LIN {X 0,Y 523.533,Z 695.705,A -85,B 0,C 180,E1 -4777.714,E2 -4777.714} C_VEL
LIN {X 0,Y 523.698,Z 688.725,A -85,B 0,C 180,E1 -4779.266,E2 -4779.266} C_VEL
LIN {X 0,Y 523.966,Z 679.973,A -85,B 0,C 180,E1 -4780.822,E2 -4780.822} C_VEL
LIN {X 0,Y 524.199,Z 670.632,A -85,B 0,C 180,E1 -4782.193,E2 -4782.193} C_VEL
LIN {X 0,Y 524.547,Z 661.185,A -85,B 0,C 180,E1 -4783.362,E2 -4783.362} C_VEL
LIN {X 0,Y 524.925,Z 649.916,A -85,B 0,C 180,E1 -4784.537,E2 -4784.537} C_VEL
LIN {X 0,Y 525.405,Z 637.565,A -85,B 0,C 180,E1 -4785.614,E2 -4785.614} C_VEL
LIN {X 0,Y 525.852,Z 623.929,A -85,B 0,C 180,E1 -4786.598,E2 -4786.598} C_VEL
LIN {X 0,Y 526.332,Z 610.529,A -85,B 0,C 180,E1 -4787.382,E2 -4787.382} C_VEL
LIN {X 0,Y 526.758,Z 595.819,A -85,B 0,C 180,E1 -4788.07,E2 -4788.07} C_VEL
LIN {X 0,Y 527.136,Z 580.489,A -85,B 0,C 180,E1 -4788.61,E2 -4788.61} C_VEL
LIN {X 0,Y 527.421,Z 564.422,A -85,B 0,C 180,E1 -4788.998,E2 -4788.998} C_VEL
LIN {X 0,Y 528.018,Z 482.561,A -85,B 0,C 180,E1 -4790.169,E2 -4790.169} C_VEL
LIN {X 0,Y 528.423,Z 411.771,A -85,B 0,C 180,E1 -4791.166,E2 -4791.166} C_VEL
LIN {X 0,Y 525.812,Z 398.27,A -85,B 0,C 180,E1 -4791.495,E2 -4791.495} C_VEL
LIN {X 0,Y 526.43,Z 378.923,A -85,B 0,C 180,E1 -4794.026,E2 -4794.026} C_VEL
LIN {X 0,Y 526.914,Z 363.166,A -85,B 0,C 180,E1 -4796.112,E2 -4796.112} C_VEL
LIN {X 0,Y 523.93,Z 349.852,A -85,B 0,C 180,E1 -4798.108,E2 -4798.108} C_VEL
LIN {X 0,Y 523.931,Z 349.846,A -85,B 0,C 180,E1 -4800.852,E2 -4800.852} C_VEL
LIN {X 0,Y 523.922,Z 349.847,A -85,B 0,C 180,E1 -4803.728,E2 -4803.728} C_VEL
LIN {X 0,Y 523.878,Z 349.856,A -85,B 0,C 180,E1 -4806.398,E2 -4806.398} C_VEL
LIN {X 0,Y 523.901,Z 349.847,A -85,B 0,C 180,E1 -4809.084,E2 -4809.084} C_VEL
LIN {X 0,Y 523.899,Z 349.854,A -85,B 0,C 180,E1 -4812.122,E2 -4812.122} C_VEL
LIN {X 0,Y 523.922,Z 349.843,A -85,B 0,C 180,E1 -4815.31,E2 -4815.31} C_VEL
LIN {X 0,Y 523.907,Z 349.847,A -85,B 0,C 180,E1 -4818.693,E2 -4818.693} C_VEL
LIN {X 0,Y 523.889,Z 349.852,A -85,B 0,C 180,E1 -4821.896,E2 -4821.896} C_VEL
LIN {X 0,Y 523.902,Z 349.845,A -85,B 0,C 180,E1 -4824.912,E2 -4824.912} C_VEL
LIN {X 0,Y 523.921,Z 349.846,A -85,B 0,C 180,E1 -4827.679,E2 -4827.679} C_VEL
LIN {X 0,Y 523.92,Z 349.845,A -85,B 0,C 180,E1 -4830.68,E2 -4830.68} C_VEL
LIN {X 0,Y 523.883,Z 349.851,A -85,B 0,C 180,E1 -4833.724,E2 -4833.724} C_VEL
LIN {X 0,Y 523.892,Z 349.853,A -85,B 0,C 180,E1 -4836.269,E2 -4836.269} C_VEL
LIN {X 0,Y 523.924,Z 349.843,A -85,B 0,C 180,E1 -4838.766,E2 -4838.766} C_VEL
LIN {X 0,Y 523.918,Z 349.843,A -85,B 0,C 180,E1 -4841.22,E2 -4841.22} C_VEL
LIN {X 0,Y 523.897,Z 349.85,A -85,B 0,C 180,E1 -4844.437,E2 -4844.437} C_VEL
LIN {X 0,Y 523.937,Z 349.844,A -85,B 0,C 180,E1 -4847.607,E2 -4847.607} C_VEL
LIN {X 0,Y 523.914,Z 349.852,A -85,B 0,C 180,E1 -4849.957,E2 -4849.957} C_VEL
LIN {X 0,Y 523.975,Z 349.836,A -85,B 0,C 180,E1 -4853.067,E2 -4853.067} C_VEL
LIN {X 0,Y 523.934,Z 349.842,A -85,B 0,C 180,E1 -4855.384,E2 -4855.384} C_VEL
LIN {X 0,Y 524.089,Z 349.826,A -85,B 0,C 180,E1 -4857.695,E2 -4857.695} C_VEL
LIN {X 0,Y 524.081,Z 349.832,A -85,B 0,C 180,E1 -4860,E2 -4860} C_VEL
LIN {X 0,Y 524.088,Z 349.826,A -85,B 0,C 180,E1 -4862.306,E2 -4862.306} C_VEL
LIN {X 0,Y 523.991,Z 349.841,A -85,B 0,C 180,E1 -4866.16,E2 -4866.16} C_VEL
LIN {X 0,Y 523.96,Z 349.839,A -85,B 0,C 180,E1 -4869.263,E2 -4869.263} C_VEL
LIN {X 0,Y 523.931,Z 349.844,A -85,B 0,C 180,E1 -4872.394,E2 -4872.394} C_VEL
LIN {X 0,Y 523.898,Z 349.849,A -85,B 0,C 180,E1 -4875.563,E2 -4875.563} C_VEL
LIN {X 0,Y 523.914,Z 349.844,A -85,B 0,C 180,E1 -4878.781,E2 -4878.781} C_VEL
LIN {X 0,Y 523.925,Z 349.843,A -85,B 0,C 180,E1 -4881.234,E2 -4881.234} C_VEL
LIN {X 0,Y 523.918,Z 349.848,A -85,B 0,C 180,E1 -4884.197,E2 -4884.197} C_VEL
LIN {X 0,Y 523.879,Z 349.848,A -85,B 0,C 180,E1 -4887.137,E2 -4887.137} C_VEL
LIN {X 0,Y 523.882,Z 349.855,A -85,B 0,C 180,E1 -4889.76,E2 -4889.76} C_VEL
LIN {X 0,Y 523.921,Z 349.844,A -85,B 0,C 180,E1 -4892.451,E2 -4892.451} C_VEL
LIN {X 0,Y 523.897,Z 349.847,A -85,B 0,C 180,E1 -4895.229,E2 -4895.229} C_VEL
LIN {X 0,Y 523.891,Z 349.852,A -85,B 0,C 180,E1 -4898.104,E2 -4898.104} C_VEL
LIN {X 0,Y 523.907,Z 349.846,A -85,B 0,C 180,E1 -4901.307,E2 -4901.307} C_VEL
LIN {X 0,Y 523.925,Z 349.842,A -85,B 0,C 180,E1 -4904.69,E2 -4904.69} C_VEL
LIN {X 0,Y 523.878,Z 349.848,A -85,B 0,C 180,E1 -4906.88,E2 -4906.88} C_VEL
LIN {X 0,Y 523.194,Z 349.94,A -85,B 0,C 180,E1 -4907.521,E2 -4907.521} C_VEL
LIN {X 0,Y 520.328,Z 350.292,A -85,B 0,C 180,E1 -4908.563,E2 -4908.563} C_VEL
LIN {X 0,Y 517.929,Z 350.592,A -85,B 0,C 180,E1 -4909.401,E2 -4909.401} C_VEL
LIN {X 0,Y 516.921,Z 350.72,A -85,B 0,C 180,E1 -4910.049,E2 -4910.049} C_VEL
LIN {X 0,Y 516.85,Z 350.726,A -85,B 0,C 180,E1 -4910.269,E2 -4910.269} C_VEL
LIN {X 0,Y 516.839,Z 350.728,A -85,B 0,C 180,E1 -4913.349,E2 -4913.349} C_VEL
LIN {X 0,Y 516.878,Z 350.724,A -85,B 0,C 180,E1 -4916.12,E2 -4916.12} C_VEL
LIN {X 0,Y 516.884,Z 350.719,A -85,B 0,C 180,E1 -4918.938,E2 -4918.938} C_VEL
LIN {X 0,Y 516.837,Z 350.732,A -85,B 0,C 180,E1 -4921.582,E2 -4921.582} C_VEL
LIN {X 0,Y 516.866,Z 350.724,A -85,B 0,C 180,E1 -4924.209,E2 -4924.209} C_VEL
LIN {X 0,Y 516.855,Z 350.723,A -85,B 0,C 180,E1 -4926.777,E2 -4926.777} C_VEL
LIN {X 0,Y 516.938,Z 350.722,A -85,B 0,C 180,E1 -4929.733,E2 -4929.733} C_VEL
LIN {X 0,Y 516.883,Z 350.719,A -85,B 0,C 180,E1 -4932.596,E2 -4932.596} C_VEL
LIN {X 0,Y 516.936,Z 350.714,A -85,B 0,C 180,E1 -4935.031,E2 -4935.031} C_VEL
LIN {X 0,Y 516.968,Z 350.711,A -85,B 0,C 180,E1 -4938.235,E2 -4938.235} C_VEL
LIN {X 0,Y 516.932,Z 350.718,A -85,B 0,C 180,E1 -4941.4,E2 -4941.4} C_VEL
LIN {X 0,Y 516.987,Z 350.707,A -85,B 0,C 180,E1 -4944.541,E2 -4944.541} C_VEL
LIN {X 0,Y 517.077,Z 350.705,A -85,B 0,C 180,E1 -4947.664,E2 -4947.664} C_VEL
LIN {X 0,Y 517.069,Z 350.7,A -85,B 0,C 180,E1 -4950.001,E2 -4950.001} C_VEL
LIN {X 0,Y 517.077,Z 350.696,A -85,B 0,C 180,E1 -4952.338,E2 -4952.338} C_VEL
LIN {X 0,Y 516.979,Z 350.709,A -85,B 0,C 180,E1 -4956.245,E2 -4956.245} C_VEL
LIN {X 0,Y 516.94,Z 350.718,A -85,B 0,C 180,E1 -4959.391,E2 -4959.391} C_VEL
LIN {X 0,Y 516.958,Z 350.716,A -85,B 0,C 180,E1 -4961.808,E2 -4961.808} C_VEL
LIN {X 0,Y 516.949,Z 350.714,A -85,B 0,C 180,E1 -4965.146,E2 -4965.146} C_VEL
LIN {X 0,Y 516.882,Z 350.721,A -85,B 0,C 180,E1 -4968.225,E2 -4968.225} C_VEL
LIN {X 0,Y 516.911,Z 350.716,A -85,B 0,C 180,E1 -4970.703,E2 -4970.703} C_VEL
LIN {X 0,Y 516.89,Z 350.721,A -85,B 0,C 180,E1 -4974.074,E2 -4974.074} C_VEL
LIN {X 0,Y 516.849,Z 350.724,A -85,B 0,C 180,E1 -4976.663,E2 -4976.663} C_VEL
LIN {X 0,Y 516.892,Z 350.727,A -85,B 0,C 180,E1 -4979.519,E2 -4979.519} C_VEL
LIN {X 0,Y 516.902,Z 350.717,A -85,B 0,C 180,E1 -4982.544,E2 -4982.544} C_VEL
LIN {X 0,Y 516.867,Z 350.728,A -85,B 0,C 180,E1 -4985.329,E2 -4985.329} C_VEL
LIN {X 0,Y 516.884,Z 350.724,A -85,B 0,C 180,E1 -4987.943,E2 -4987.943} C_VEL
LIN {X 0,Y 516.878,Z 350.723,A -85,B 0,C 180,E1 -4990.743,E2 -4990.743} C_VEL
LIN {X 0,Y 516.887,Z 350.727,A -85,B 0,C 180,E1 -4993.893,E2 -4993.893} C_VEL
LIN {X 0,Y 516.924,Z 350.853,A -85,B 0,C 180,E1 -4996.033,E2 -4996.033} C_VEL
LIN {X 0,Y 518.959,Z 360.312,A -85,B 0,C 180,E1 -4997.639,E2 -4997.639} C_VEL
LIN {X 0,Y 518.787,Z 370.855,A -85,B 0,C 180,E1 -4999.267,E2 -4999.267} C_VEL
LIN {X 0,Y 521.906,Z 385.017,A -85,B 0,C 180,E1 -4999.622,E2 -4999.622} C_VEL
LIN {X 0,Y 520.71,Z 536.608,A -85,B 0,C 180,E1 -5001.836,E2 -5001.836} C_VEL
LIN {X 0,Y 520.403,Z 552.083,A -85,B 0,C 180,E1 -5002.224,E2 -5002.224} C_VEL
LIN {X 0,Y 519.996,Z 566.356,A -85,B 0,C 180,E1 -5002.733,E2 -5002.733} C_VEL
LIN {X 0,Y 519.561,Z 580.137,A -85,B 0,C 180,E1 -5003.38,E2 -5003.38} C_VEL
LIN {X 0,Y 519.167,Z 592.322,A -85,B 0,C 180,E1 -5004.09,E2 -5004.09} C_VEL
LIN {X 0,Y 518.645,Z 604.733,A -85,B 0,C 180,E1 -5004.955,E2 -5004.955} C_VEL
LIN {X 0,Y 518.169,Z 617.851,A -85,B 0,C 180,E1 -5006.069,E2 -5006.069} C_VEL
LIN {X 0,Y 517.742,Z 628.127,A -85,B 0,C 180,E1 -5007.113,E2 -5007.113} C_VEL
LIN {X 0,Y 517.366,Z 637.65,A -85,B 0,C 180,E1 -5008.238,E2 -5008.238} C_VEL
LIN {X 0,Y 517.032,Z 647.144,A -85,B 0,C 180,E1 -5009.579,E2 -5009.579} C_VEL
LIN {X 0,Y 516.749,Z 655.098,A -85,B 0,C 180,E1 -5010.908,E2 -5010.908} C_VEL
LIN {X 0,Y 516.536,Z 662.608,A -85,B 0,C 180,E1 -5012.444,E2 -5012.444} C_VEL
LIN {X 0,Y 516.42,Z 668.488,A -85,B 0,C 180,E1 -5013.923,E2 -5013.923} C_VEL
LIN {X 0,Y 516.306,Z 673.209,A -85,B 0,C 180,E1 -5015.455,E2 -5015.455} C_VEL
LIN {X 0,Y 516.214,Z 676.291,A -85,B 0,C 180,E1 -5016.745,E2 -5016.745} C_VEL
LIN {X 0,Y 516.181,Z 678.984,A -85,B 0,C 180,E1 -5018.431,E2 -5018.431} C_VEL
LIN {X 0,Y 516.199,Z 680.402,A -85,B 0,C 180,E1 -5020.1,E2 -5020.1} C_VEL
LIN {X 0,Y 516.165,Z 680.465,A -85,B 0,C 180,E1 -5021.75,E2 -5021.75} C_VEL
LIN {X 0,Y 516.169,Z 679.334,A -85,B 0,C 180,E1 -5023.385,E2 -5023.385} C_VEL
LIN {X 0,Y 516.212,Z 676.933,A -85,B 0,C 180,E1 -5025.008,E2 -5025.008} C_VEL
LIN {X 0,Y 516.279,Z 673.27,A -85,B 0,C 180,E1 -5026.619,E2 -5026.619} C_VEL
LIN {X 0,Y 516.387,Z 668.327,A -85,B 0,C 180,E1 -5028.22,E2 -5028.22} C_VEL
LIN {X 0,Y 516.557,Z 661.89,A -85,B 0,C 180,E1 -5029.812,E2 -5029.812} C_VEL
LIN {X 0,Y 516.8,Z 653.92,A -85,B 0,C 180,E1 -5031.397,E2 -5031.397} C_VEL
LIN {X 0,Y 517.106,Z 645.168,A -85,B 0,C 180,E1 -5032.817,E2 -5032.817} C_VEL
LIN {X 0,Y 517.457,Z 635.233,A -85,B 0,C 180,E1 -5034.153,E2 -5034.153} C_VEL
LIN {X 0,Y 517.851,Z 624.884,A -85,B 0,C 180,E1 -5035.329,E2 -5035.329} C_VEL
LIN {X 0,Y 518.291,Z 613.595,A -85,B 0,C 180,E1 -5036.404,E2 -5036.404} C_VEL
LIN {X 0,Y 518.823,Z 601.429,A -85,B 0,C 180,E1 -5037.379,E2 -5037.379} C_VEL
LIN {X 0,Y 519.301,Z 588.182,A -85,B 0,C 180,E1 -5038.255,E2 -5038.255} C_VEL
LIN {X 0,Y 519.79,Z 573.497,A -85,B 0,C 180,E1 -5039.031,E2 -5039.031} C_VEL
LIN {X 0,Y 520.184,Z 558.316,A -85,B 0,C 180,E1 -5039.648,E2 -5039.648} C_VEL
LIN {X 0,Y 520.543,Z 542.685,A -85,B 0,C 180,E1 -5040.103,E2 -5040.103} C_VEL
LIN {X 0,Y 520.711,Z 526.129,A -85,B 0,C 180,E1 -5040.409,E2 -5040.409} C_VEL
LIN {X 0,Y 521.891,Z 388.15,A -85,B 0,C 180,E1 -5042.421,E2 -5042.421} C_VEL
LIN {X 0,Y 521.675,Z 383.753,A -85,B 0,C 180,E1 -5042.499,E2 -5042.499} C_VEL
LIN {X 0,Y 518.92,Z 371.346,A -85,B 0,C 180,E1 -5042.821,E2 -5042.821} C_VEL
LIN {X 0,Y 519.16,Z 360.873,A -85,B 0,C 180,E1 -5044.464,E2 -5044.464} C_VEL
LIN {X 0,Y 517.011,Z 350.712,A -85,B 0,C 180,E1 -5046.243,E2 -5046.243} C_VEL
LIN {X 0,Y 516.942,Z 350.718,A -85,B 0,C 180,E1 -5049.389,E2 -5049.389} C_VEL
LIN {X 0,Y 516.957,Z 350.713,A -85,B 0,C 180,E1 -5051.807,E2 -5051.807} C_VEL
LIN {X 0,Y 516.949,Z 350.716,A -85,B 0,C 180,E1 -5055.146,E2 -5055.146} C_VEL
LIN {X 0,Y 516.916,Z 350.724,A -85,B 0,C 180,E1 -5058.222,E2 -5058.222} C_VEL
LIN {X 0,Y 516.916,Z 350.721,A -85,B 0,C 180,E1 -5060.701,E2 -5060.701} C_VEL
LIN {X 0,Y 516.888,Z 350.726,A -85,B 0,C 180,E1 -5064.073,E2 -5064.073} C_VEL
LIN {X 0,Y 516.839,Z 350.731,A -85,B 0,C 180,E1 -5066.662,E2 -5066.662} C_VEL
LIN {X 0,Y 516.888,Z 350.722,A -85,B 0,C 180,E1 -5069.518,E2 -5069.518} C_VEL
LIN {X 0,Y 516.893,Z 350.724,A -85,B 0,C 180,E1 -5072.542,E2 -5072.542} C_VEL
LIN {X 0,Y 516.851,Z 350.726,A -85,B 0,C 180,E1 -5075.326,E2 -5075.326} C_VEL
LIN {X 0,Y 516.871,Z 350.724,A -85,B 0,C 180,E1 -5078.717,E2 -5078.717} C_VEL
LIN {X 0,Y 516.834,Z 350.732,A -85,B 0,C 180,E1 -5081.783,E2 -5081.783} C_VEL
LIN {X 0,Y 516.899,Z 350.718,A -85,B 0,C 180,E1 -5085.006,E2 -5085.006} C_VEL
LIN {X 0,Y 516.831,Z 350.73,A -85,B 0,C 180,E1 -5088.409,E2 -5088.409} C_VEL
LIN {X 0,Y 516.861,Z 350.726,A -85,B 0,C 180,E1 -5091.281,E2 -5091.281} C_VEL
LIN {X 0,Y 516.829,Z 350.731,A -85,B 0,C 180,E1 -5094.676,E2 -5094.676} C_VEL
LIN {X 0,Y 516.866,Z 350.731,A -85,B 0,C 180,E1 -5097.462,E2 -5097.462} C_VEL
LIN {X 0,Y 516.887,Z 350.727,A -85,B 0,C 180,E1 -5100.481,E2 -5100.481} C_VEL
LIN {X 0,Y 516.857,Z 350.743,A -85,B 0,C 180,E1 -5101.725,E2 -5101.725} C_VEL
LIN {X 0,Y 519.892,Z 363.888,A -85,B 0,C 180,E1 -5103.721,E2 -5103.721} C_VEL
LIN {X 0,Y 519.532,Z 376.499,A -85,B 0,C 180,E1 -5105.418,E2 -5105.418} C_VEL
LIN {X 0,Y 518.912,Z 397.028,A -85,B 0,C 180,E1 -5108.133,E2 -5108.133} C_VEL
LIN {X 0,Y 518.86,Z 397.663,A -85,B 0,C 180,E1 -5108.214,E2 -5108.214} C_VEL
LIN {X 0,Y 521.848,Z 413.736,A -85,B 0,C 180,E1 -5108.593,E2 -5108.593} C_VEL
LIN {X 0,Y 520.618,Z 564.199,A -85,B 0,C 180,E1 -5110.789,E2 -5110.789} C_VEL
LIN {X 0,Y 520.325,Z 579.46,A -85,B 0,C 180,E1 -5111.159,E2 -5111.159} C_VEL
LIN {X 0,Y 519.993,Z 593.147,A -85,B 0,C 180,E1 -5111.633,E2 -5111.633} C_VEL
LIN {X 0,Y 519.517,Z 607.479,A -85,B 0,C 180,E1 -5112.278,E2 -5112.278} C_VEL
LIN {X 0,Y 519.019,Z 621.427,A -85,B 0,C 180,E1 -5113.073,E2 -5113.073} C_VEL
LIN {X 0,Y 518.575,Z 634.218,A -85,B 0,C 180,E1 -5113.97,E2 -5113.97} C_VEL
LIN {X 0,Y 518.12,Z 645.2,A -85,B 0,C 180,E1 -5114.883,E2 -5114.883} C_VEL
LIN {X 0,Y 517.681,Z 657.06,A -85,B 0,C 180,E1 -5116.055,E2 -5116.055} C_VEL
LIN {X 0,Y 517.288,Z 667.206,A -85,B 0,C 180,E1 -5117.244,E2 -5117.244} C_VEL
LIN {X 0,Y 516.933,Z 677.106,A -85,B 0,C 180,E1 -5118.63,E2 -5118.63} C_VEL
LIN {X 0,Y 516.678,Z 685.348,A -85,B 0,C 180,E1 -5120.012,E2 -5120.012} C_VEL
LIN {X 0,Y 516.541,Z 692.142,A -85,B 0,C 180,E1 -5121.391,E2 -5121.391} C_VEL
LIN {X 0,Y 516.392,Z 698.414,A -85,B 0,C 180,E1 -5122.963,E2 -5122.963} C_VEL
LIN {X 0,Y 516.352,Z 703.261,A -85,B 0,C 180,E1 -5124.532,E2 -5124.532} C_VEL
LIN {X 0,Y 516.293,Z 706.806,A -85,B 0,C 180,E1 -5126.096,E2 -5126.096} C_VEL
LIN {X 0,Y 516.258,Z 709.135,A -85,B 0,C 180,E1 -5127.658,E2 -5127.658} C_VEL
LIN {X 0,Y 516.156,Z 710.305,A -85,B 0,C 180,E1 -5129.219,E2 -5129.219} C_VEL
LIN {X 0,Y 516.156,Z 710.305,A -85,B 0,C 180,E1 -5130.779,E2 -5130.779} C_VEL
LIN {X 0,Y 516.258,Z 709.135,A -85,B 0,C 180,E1 -5132.339,E2 -5132.339} C_VEL
LIN {X 0,Y 516.307,Z 706.811,A -85,B 0,C 180,E1 -5133.901,E2 -5133.901} C_VEL
LIN {X 0,Y 516.352,Z 703.279,A -85,B 0,C 180,E1 -5135.466,E2 -5135.466} C_VEL
LIN {X 0,Y 516.394,Z 698.447,A -85,B 0,C 180,E1 -5137.034,E2 -5137.034} C_VEL
LIN {X 0,Y 516.539,Z 692.184,A -85,B 0,C 180,E1 -5138.606,E2 -5138.606} C_VEL
LIN {X 0,Y 516.727,Z 684.306,A -85,B 0,C 180,E1 -5140.183,E2 -5140.183} C_VEL
LIN {X 0,Y 516.996,Z 675.916,A -85,B 0,C 180,E1 -5141.565,E2 -5141.565} C_VEL
LIN {X 0,Y 517.381,Z 665.795,A -85,B 0,C 180,E1 -5142.951,E2 -5142.951} C_VEL
LIN {X 0,Y 517.737,Z 655.446,A -85,B 0,C 180,E1 -5144.141,E2 -5144.141} C_VEL
LIN {X 0,Y 518.227,Z 643.429,A -85,B 0,C 180,E1 -5145.301,E2 -5145.301} C_VEL
LIN {X 0,Y 518.713,Z 630.654,A -85,B 0,C 180,E1 -5146.327,E2 -5146.327} C_VEL
LIN {X 0,Y 519.29,Z 617.094,A -85,B 0,C 180,E1 -5147.219,E2 -5147.219} C_VEL
LIN {X 0,Y 519.73,Z 602.03,A -85,B 0,C 180,E1 -5148.017,E2 -5148.017} C_VEL
LIN {X 0,Y 520.207,Z 586.653,A -85,B 0,C 180,E1 -5148.637,E2 -5148.637} C_VEL
LIN {X 0,Y 520.527,Z 571.093,A -85,B 0,C 180,E1 -5149.09,E2 -5149.09} C_VEL
LIN {X 0,Y 520.763,Z 554.696,A -85,B 0,C 180,E1 -5149.392,E2 -5149.392} C_VEL
LIN {X 0,Y 521.852,Z 413.102,A -85,B 0,C 180,E1 -5151.423,E2 -5151.423} C_VEL
LIN {X 0,Y 518.96,Z 398.158,A -85,B 0,C 180,E1 -5151.785,E2 -5151.785} C_VEL
LIN {X 0,Y 519.601,Z 378.766,A -85,B 0,C 180,E1 -5154.363,E2 -5154.363} C_VEL
LIN {X 0,Y 520.056,Z 364.594,A -85,B 0,C 180,E1 -5156.267,E2 -5156.267} C_VEL
LIN {X 0,Y 516.884,Z 350.729,A -85,B 0,C 180,E1 -5158.382,E2 -5158.382} C_VEL
LIN {X 0,Y 516.88,Z 350.724,A -85,B 0,C 180,E1 -5161.108,E2 -5161.108} C_VEL
LIN {X 0,Y 516.877,Z 350.727,A -85,B 0,C 180,E1 -5163.961,E2 -5163.961} C_VEL
LIN {X 0,Y 516.834,Z 350.729,A -85,B 0,C 180,E1 -5166.748,E2 -5166.748} C_VEL
LIN {X 0,Y 516.847,Z 350.728,A -85,B 0,C 180,E1 -5169.722,E2 -5169.722} C_VEL
LIN {X 0,Y 516.873,Z 350.724,A -85,B 0,C 180,E1 -5171.777,E2 -5171.777} C_VEL
LIN {X 0,Y 516.884,Z 350.72,A -85,B 0,C 180,E1 -5175.006,E2 -5175.006} C_VEL
LIN {X 0,Y 516.843,Z 350.73,A -85,B 0,C 180,E1 -5178.405,E2 -5178.405} C_VEL
LIN {X 0,Y 516.86,Z 350.722,A -85,B 0,C 180,E1 -5181.282,E2 -5181.282} C_VEL
LIN {X 0,Y 516.839,Z 350.727,A -85,B 0,C 180,E1 -5184.672,E2 -5184.672} C_VEL
LIN {X 0,Y 516.881,Z 350.721,A -85,B 0,C 180,E1 -5187.456,E2 -5187.456} C_VEL
LIN {X 0,Y 516.888,Z 350.72,A -85,B 0,C 180,E1 -5190.694,E2 -5190.694} C_VEL
LIN {X 0,Y 516.863,Z 350.727,A -85,B 0,C 180,E1 -5193.818,E2 -5193.818} C_VEL
LIN {X 0,Y 516.841,Z 350.726,A -85,B 0,C 180,E1 -5196.775,E2 -5196.775} C_VEL
LIN {X 0,Y 516.913,Z 350.72,A -85,B 0,C 180,E1 -5199.735,E2 -5199.735} C_VEL
LIN {X 0,Y 516.852,Z 350.725,A -85,B 0,C 180,E1 -5202.594,E2 -5202.594} C_VEL
LIN {X 0,Y 516.919,Z 350.715,A -85,B 0,C 180,E1 -5205.03,E2 -5205.03} C_VEL
LIN {X 0,Y 516.951,Z 350.717,A -85,B 0,C 180,E1 -5208.234,E2 -5208.234} C_VEL
LIN {X 0,Y 516.917,Z 350.716,A -85,B 0,C 180,E1 -5211.399,E2 -5211.399} C_VEL
LIN {X 0,Y 516.973,Z 350.71,A -85,B 0,C 180,E1 -5214.54,E2 -5214.54} C_VEL
LIN {X 0,Y 517.058,Z 350.702,A -85,B 0,C 180,E1 -5217.663,E2 -5217.663} C_VEL
LIN {X 0,Y 517.05,Z 350.708,A -85,B 0,C 180,E1 -5220,E2 -5220} C_VEL
LIN {X 0,Y 517.058,Z 350.702,A -85,B 0,C 180,E1 -5222.337,E2 -5222.337} C_VEL
LIN {X 0,Y 516.957,Z 350.715,A -85,B 0,C 180,E1 -5226.244,E2 -5226.244} C_VEL
LIN {X 0,Y 516.915,Z 350.717,A -85,B 0,C 180,E1 -5229.39,E2 -5229.39} C_VEL
LIN {X 0,Y 516.884,Z 350.721,A -85,B 0,C 180,E1 -5232.565,E2 -5232.565} C_VEL
LIN {X 0,Y 516.924,Z 350.715,A -85,B 0,C 180,E1 -5235.144,E2 -5235.144} C_VEL
LIN {X 0,Y 516.861,Z 350.727,A -85,B 0,C 180,E1 -5238.225,E2 -5238.225} C_VEL
LIN {X 0,Y 516.885,Z 350.72,A -85,B 0,C 180,E1 -5240.703,E2 -5240.703} C_VEL
LIN {X 0,Y 516.842,Z 350.725,A -85,B 0,C 180,E1 -5243.225,E2 -5243.225} C_VEL
LIN {X 0,Y 516.864,Z 350.727,A -85,B 0,C 180,E1 -5246.182,E2 -5246.182} C_VEL
LIN {X 0,Y 516.872,Z 350.725,A -85,B 0,C 180,E1 -5249.52,E2 -5249.52} C_VEL
LIN {X 0,Y 516.883,Z 350.72,A -85,B 0,C 180,E1 -5252.544,E2 -5252.544} C_VEL
LIN {X 0,Y 516.841,Z 350.727,A -85,B 0,C 180,E1 -5255.329,E2 -5255.329} C_VEL
LIN {X 0,Y 516.862,Z 350.722,A -85,B 0,C 180,E1 -5258.718,E2 -5258.718} C_VEL
LIN {X 0,Y 516.838,Z 350.734,A -85,B 0,C 180,E1 -5261.783,E2 -5261.783} C_VEL
LIN {X 0,Y 516.887,Z 350.719,A -85,B 0,C 180,E1 -5265.008,E2 -5265.008} C_VEL
LIN {X 0,Y 516.878,Z 350.722,A -85,B 0,C 180,E1 -5268.404,E2 -5268.404} C_VEL
LIN {X 0,Y 516.85,Z 350.726,A -85,B 0,C 180,E1 -5270.269,E2 -5270.269} C_VEL
LIN {X 0,Y 516.212,Z 350.808,A -85,B 0,C 180,E1 -5270.919,E2 -5270.919} C_VEL
LIN {X 0,Y 513.364,Z 351.17,A -85,B 0,C 180,E1 -5271.974,E2 -5271.974} C_VEL
LIN {X 0,Y 510.934,Z 351.474,A -85,B 0,C 180,E1 -5272.824,E2 -5272.824} C_VEL
LIN {X 0,Y 509.882,Z 351.6,A -85,B 0,C 180,E1 -5273.481,E2 -5273.481} C_VEL
LIN {X 0,Y 509.794,Z 351.609,A -85,B 0,C 180,E1 -5273.703,E2 -5273.703} C_VEL
LIN {X 0,Y 509.836,Z 351.598,A -85,B 0,C 180,E1 -5276.539,E2 -5276.539} C_VEL
LIN {X 0,Y 509.829,Z 351.601,A -85,B 0,C 180,E1 -5279.335,E2 -5279.335} C_VEL
LIN {X 0,Y 509.821,Z 351.604,A -85,B 0,C 180,E1 -5282.052,E2 -5282.052} C_VEL
LIN {X 0,Y 509.798,Z 351.602,A -85,B 0,C 180,E1 -5284.701,E2 -5284.701} C_VEL
LIN {X 0,Y 509.824,Z 351.604,A -85,B 0,C 180,E1 -5287.46,E2 -5287.46} C_VEL
LIN {X 0,Y 509.915,Z 351.595,A -85,B 0,C 180,E1 -5289.846,E2 -5289.846} C_VEL
LIN {X 0,Y 509.851,Z 351.597,A -85,B 0,C 180,E1 -5293.175,E2 -5293.175} C_VEL
LIN {X 0,Y 509.853,Z 351.603,A -85,B 0,C 180,E1 -5295.635,E2 -5295.635} C_VEL
LIN {X 0,Y 509.912,Z 351.588,A -85,B 0,C 180,E1 -5298.876,E2 -5298.876} C_VEL
LIN {X 0,Y 509.878,Z 351.595,A -85,B 0,C 180,E1 -5302.079,E2 -5302.079} C_VEL
LIN {X 0,Y 509.942,Z 351.584,A -85,B 0,C 180,E1 -5304.465,E2 -5304.465} C_VEL
LIN {X 0,Y 510.045,Z 351.58,A -85,B 0,C 180,E1 -5307.632,E2 -5307.632} C_VEL
LIN {X 0,Y 510.038,Z 351.576,A -85,B 0,C 180,E1 -5310.001,E2 -5310.001} C_VEL
LIN {X 0,Y 510.046,Z 351.572,A -85,B 0,C 180,E1 -5312.37,E2 -5312.37} C_VEL
LIN {X 0,Y 509.944,Z 351.592,A -85,B 0,C 180,E1 -5315.537,E2 -5315.537} C_VEL
LIN {X 0,Y 509.905,Z 351.589,A -85,B 0,C 180,E1 -5318.721,E2 -5318.721} C_VEL
LIN {X 0,Y 509.91,Z 351.592,A -85,B 0,C 180,E1 -5321.933,E2 -5321.933} C_VEL
LIN {X 0,Y 509.901,Z 351.593,A -85,B 0,C 180,E1 -5325.243,E2 -5325.243} C_VEL
LIN {X 0,Y 509.842,Z 351.597,A -85,B 0,C 180,E1 -5328.485,E2 -5328.485} C_VEL
LIN {X 0,Y 509.852,Z 351.597,A -85,B 0,C 180,E1 -5331.003,E2 -5331.003} C_VEL
LIN {X 0,Y 509.824,Z 351.608,A -85,B 0,C 180,E1 -5333.565,E2 -5333.565} C_VEL
LIN {X 0,Y 509.824,Z 351.599,A -85,B 0,C 180,E1 -5336.358,E2 -5336.358} C_VEL
LIN {X 0,Y 509.844,Z 351.597,A -85,B 0,C 180,E1 -5338.847,E2 -5338.847} C_VEL
LIN {X 0,Y 509.825,Z 351.607,A -85,B 0,C 180,E1 -5341.591,E2 -5341.591} C_VEL
LIN {X 0,Y 509.846,Z 351.596,A -85,B 0,C 180,E1 -5344.415,E2 -5344.415} C_VEL
LIN {X 0,Y 509.814,Z 351.609,A -85,B 0,C 180,E1 -5347.342,E2 -5347.342} C_VEL
LIN {X 0,Y 509.839,Z 351.6,A -85,B 0,C 180,E1 -5350.383,E2 -5350.383} C_VEL
LIN {X 0,Y 509.81,Z 351.607,A -85,B 0,C 180,E1 -5353.06,E2 -5353.06} C_VEL
LIN {X 0,Y 509.885,Z 351.755,A -85,B 0,C 180,E1 -5355.787,E2 -5355.787} C_VEL
LIN {X 0,Y 512.03,Z 361.637,A -85,B 0,C 180,E1 -5357.489,E2 -5357.489} C_VEL
LIN {X 0,Y 512.036,Z 369.874,A -85,B 0,C 180,E1 -5358.789,E2 -5358.789} C_VEL
LIN {X 0,Y 511.997,Z 371.041,A -85,B 0,C 180,E1 -5358.966,E2 -5358.966} C_VEL
LIN {X 0,Y 515.29,Z 385.816,A -85,B 0,C 180,E1 -5359.345,E2 -5359.345} C_VEL
LIN {X 0,Y 513.978,Z 536.633,A -85,B 0,C 180,E1 -5361.588,E2 -5361.588} C_VEL
LIN {X 0,Y 513.639,Z 552.101,A -85,B 0,C 180,E1 -5361.979,E2 -5361.979} C_VEL
LIN {X 0,Y 513.205,Z 567.388,A -85,B 0,C 180,E1 -5362.537,E2 -5362.537} C_VEL
LIN {X 0,Y 512.725,Z 581.415,A -85,B 0,C 180,E1 -5363.213,E2 -5363.213} C_VEL
LIN {X 0,Y 512.22,Z 595.245,A -85,B 0,C 180,E1 -5364.05,E2 -5364.05} C_VEL
LIN {X 0,Y 511.638,Z 608.164,A -85,B 0,C 180,E1 -5365.007,E2 -5365.007} C_VEL
LIN {X 0,Y 511.146,Z 619.76,A -85,B 0,C 180,E1 -5366.042,E2 -5366.042} C_VEL
LIN {X 0,Y 510.676,Z 630.854,A -85,B 0,C 180,E1 -5367.222,E2 -5367.222} C_VEL
LIN {X 0,Y 510.282,Z 640.539,A -85,B 0,C 180,E1 -5368.441,E2 -5368.441} C_VEL
LIN {X 0,Y 509.942,Z 649.621,A -85,B 0,C 180,E1 -5369.798,E2 -5369.798} C_VEL
LIN {X 0,Y 509.65,Z 657.133,A -85,B 0,C 180,E1 -5371.141,E2 -5371.141} C_VEL
LIN {X 0,Y 509.465,Z 663.421,A -85,B 0,C 180,E1 -5372.475,E2 -5372.475} C_VEL
LIN {X 0,Y 509.343,Z 668.555,A -85,B 0,C 180,E1 -5373.797,E2 -5373.797} C_VEL
LIN {X 0,Y 509.245,Z 672.646,A -85,B 0,C 180,E1 -5375.107,E2 -5375.107} C_VEL
LIN {X 0,Y 509.141,Z 675.85,A -85,B 0,C 180,E1 -5376.402,E2 -5376.402} C_VEL
LIN {X 0,Y 509.089,Z 678.85,A -85,B 0,C 180,E1 -5378.115,E2 -5378.115} C_VEL
LIN {X 0,Y 509.092,Z 680.479,A -85,B 0,C 180,E1 -5379.842,E2 -5379.842} C_VEL
LIN {X 0,Y 509.084,Z 680.745,A -85,B 0,C 180,E1 -5381.487,E2 -5381.487} C_VEL
LIN {X 0,Y 509.082,Z 679.824,A -85,B 0,C 180,E1 -5383.147,E2 -5383.147} C_VEL
LIN {X 0,Y 509.111,Z 677.606,A -85,B 0,C 180,E1 -5384.794,E2 -5384.794} C_VEL
LIN {X 0,Y 509.171,Z 674.181,A -85,B 0,C 180,E1 -5386.429,E2 -5386.429} C_VEL
LIN {X 0,Y 509.318,Z 669.393,A -85,B 0,C 180,E1 -5388.054,E2 -5388.054} C_VEL
LIN {X 0,Y 509.47,Z 663.231,A -85,B 0,C 180,E1 -5389.669,E2 -5389.669} C_VEL
LIN {X 0,Y 509.702,Z 655.523,A -85,B 0,C 180,E1 -5391.276,E2 -5391.276} C_VEL
LIN {X 0,Y 510.057,Z 646.553,A -85,B 0,C 180,E1 -5392.787,E2 -5392.787} C_VEL
LIN {X 0,Y 510.396,Z 637.422,A -85,B 0,C 180,E1 -5394.072,E2 -5394.072} C_VEL
LIN {X 0,Y 510.809,Z 627.352,A -85,B 0,C 180,E1 -5395.265,E2 -5395.265} C_VEL
LIN {X 0,Y 511.315,Z 615.421,A -85,B 0,C 180,E1 -5396.454,E2 -5396.454} C_VEL
LIN {X 0,Y 511.927,Z 602.204,A -85,B 0,C 180,E1 -5397.541,E2 -5397.541} C_VEL
LIN {X 0,Y 512.426,Z 589.05,A -85,B 0,C 180,E1 -5398.428,E2 -5398.428} C_VEL
LIN {X 0,Y 512.948,Z 574.539,A -85,B 0,C 180,E1 -5399.215,E2 -5399.215} C_VEL
LIN {X 0,Y 513.39,Z 560.076,A -85,B 0,C 180,E1 -5399.822,E2 -5399.822} C_VEL
LIN {X 0,Y 513.756,Z 544.745,A -85,B 0,C 180,E1 -5400.294,E2 -5400.294} C_VEL
LIN {X 0,Y 513.942,Z 529.797,A -85,B 0,C 180,E1 -5400.597,E2 -5400.597} C_VEL
LIN {X 0,Y 515.274,Z 387.204,A -85,B 0,C 180,E1 -5402.721,E2 -5402.721} C_VEL
LIN {X 0,Y 514.659,Z 382.848,A -85,B 0,C 180,E1 -5402.817,E2 -5402.817} C_VEL
LIN {X 0,Y 512.107,Z 371.637,A -85,B 0,C 180,E1 -5403.127,E2 -5403.127} C_VEL
LIN {X 0,Y 512.351,Z 362.839,A -85,B 0,C 180,E1 -5404.524,E2 -5404.524} C_VEL
LIN {X 0,Y 509.977,Z 351.588,A -85,B 0,C 180,E1 -5406.533,E2 -5406.533} C_VEL
LIN {X 0,Y 509.883,Z 351.597,A -85,B 0,C 180,E1 -5409.52,E2 -5409.52} C_VEL
LIN {X 0,Y 509.909,Z 351.592,A -85,B 0,C 180,E1 -5411.931,E2 -5411.931} C_VEL
LIN {X 0,Y 509.899,Z 351.594,A -85,B 0,C 180,E1 -5415.241,E2 -5415.241} C_VEL
LIN {X 0,Y 509.861,Z 351.603,A -85,B 0,C 180,E1 -5418.484,E2 -5418.484} C_VEL
LIN {X 0,Y 509.854,Z 351.598,A -85,B 0,C 180,E1 -5421.001,E2 -5421.001} C_VEL
LIN {X 0,Y 509.822,Z 351.602,A -85,B 0,C 180,E1 -5423.564,E2 -5423.564} C_VEL
LIN {X 0,Y 509.817,Z 351.608,A -85,B 0,C 180,E1 -5426.356,E2 -5426.356} C_VEL
LIN {X 0,Y 509.836,Z 351.601,A -85,B 0,C 180,E1 -5428.847,E2 -5428.847} C_VEL
LIN {X 0,Y 509.814,Z 351.602,A -85,B 0,C 180,E1 -5431.59,E2 -5431.59} C_VEL
LIN {X 0,Y 509.836,Z 351.605,A -85,B 0,C 180,E1 -5434.414,E2 -5434.414} C_VEL
LIN {X 0,Y 509.78,Z 351.606,A -85,B 0,C 180,E1 -5437.344,E2 -5437.344} C_VEL
LIN {X 0,Y 509.789,Z 351.61,A -85,B 0,C 180,E1 -5440.387,E2 -5440.387} C_VEL
LIN {X 0,Y 509.793,Z 351.606,A -85,B 0,C 180,E1 -5443.574,E2 -5443.574} C_VEL
LIN {X 0,Y 509.793,Z 351.607,A -85,B 0,C 180,E1 -5446.424,E2 -5446.424} C_VEL
LIN {X 0,Y 509.788,Z 351.608,A -85,B 0,C 180,E1 -5449.612,E2 -5449.612} C_VEL
LIN {X 0,Y 509.776,Z 351.609,A -85,B 0,C 180,E1 -5452.655,E2 -5452.655} C_VEL
LIN {X 0,Y 509.831,Z 351.608,A -85,B 0,C 180,E1 -5455.802,E2 -5455.802} C_VEL
LIN {X 0,Y 509.837,Z 351.605,A -85,B 0,C 180,E1 -5458.722,E2 -5458.722} C_VEL
LIN {X 0,Y 509.831,Z 351.694,A -85,B 0,C 180,E1 -5461.448,E2 -5461.448} C_VEL
LIN {X 0,Y 513.007,Z 365.312,A -85,B 0,C 180,E1 -5463.56,E2 -5463.56} C_VEL
LIN {X 0,Y 512.825,Z 374.71,A -85,B 0,C 180,E1 -5464.859,E2 -5464.859} C_VEL
LIN {X 0,Y 512.083,Z 395.346,A -85,B 0,C 180,E1 -5467.634,E2 -5467.634} C_VEL
LIN {X 0,Y 512.059,Z 397.604,A -85,B 0,C 180,E1 -5467.914,E2 -5467.914} C_VEL
LIN {X 0,Y 515.227,Z 414.265,A -85,B 0,C 180,E1 -5468.317,E2 -5468.317} C_VEL
LIN {X 0,Y 513.838,Z 564.042,A -85,B 0,C 180,E1 -5470.551,E2 -5470.551} C_VEL
LIN {X 0,Y 513.515,Z 579.999,A -85,B 0,C 180,E1 -5470.949,E2 -5470.949} C_VEL
LIN {X 0,Y 513.107,Z 595.05,A -85,B 0,C 180,E1 -5471.49,E2 -5471.49} C_VEL
LIN {X 0,Y 512.609,Z 608.762,A -85,B 0,C 180,E1 -5472.135,E2 -5472.135} C_VEL
LIN {X 0,Y 512.077,Z 622.408,A -85,B 0,C 180,E1 -5472.94,E2 -5472.94} C_VEL
LIN {X 0,Y 511.604,Z 634.982,A -85,B 0,C 180,E1 -5473.847,E2 -5473.847} C_VEL
LIN {X 0,Y 511.011,Z 647.754,A -85,B 0,C 180,E1 -5474.953,E2 -5474.953} C_VEL
LIN {X 0,Y 510.623,Z 658.438,A -85,B 0,C 180,E1 -5476.062,E2 -5476.062} C_VEL
LIN {X 0,Y 510.21,Z 668.324,A -85,B 0,C 180,E1 -5477.267,E2 -5477.267} C_VEL
LIN {X 0,Y 509.854,Z 678.162,A -85,B 0,C 180,E1 -5478.696,E2 -5478.696} C_VEL
LIN {X 0,Y 509.577,Z 686.057,A -85,B 0,C 180,E1 -5480.072,E2 -5480.072} C_VEL
LIN {X 0,Y 509.413,Z 693.557,A -85,B 0,C 180,E1 -5481.67,E2 -5481.67} C_VEL
LIN {X 0,Y 509.29,Z 699.497,A -85,B 0,C 180,E1 -5483.263,E2 -5483.263} C_VEL
LIN {X 0,Y 509.267,Z 703.016,A -85,B 0,C 180,E1 -5484.455,E2 -5484.455} C_VEL
LIN {X 0,Y 509.187,Z 706.578,A -85,B 0,C 180,E1 -5486.042,E2 -5486.042} C_VEL
LIN {X 0,Y 509.186,Z 708.922,A -85,B 0,C 180,E1 -5487.626,E2 -5487.626} C_VEL
LIN {X 0,Y 509.07,Z 710.098,A -85,B 0,C 180,E1 -5489.208,E2 -5489.208} C_VEL
LIN {X 0,Y 509.069,Z 710.101,A -85,B 0,C 180,E1 -5490.79,E2 -5490.79} C_VEL
LIN {X 0,Y 509.186,Z 708.93,A -85,B 0,C 180,E1 -5492.372,E2 -5492.372} C_VEL
LIN {X 0,Y 509.2,Z 706.599,A -85,B 0,C 180,E1 -5493.956,E2 -5493.956} C_VEL
LIN {X 0,Y 509.267,Z 703.058,A -85,B 0,C 180,E1 -5495.542,E2 -5495.542} C_VEL
LIN {X 0,Y 509.316,Z 698.212,A -85,B 0,C 180,E1 -5497.133,E2 -5497.133} C_VEL
LIN {X 0,Y 509.477,Z 691.93,A -85,B 0,C 180,E1 -5498.726,E2 -5498.726} C_VEL
LIN {X 0,Y 509.681,Z 684.031,A -85,B 0,C 180,E1 -5500.325,E2 -5500.325} C_VEL
LIN {X 0,Y 509.963,Z 675.358,A -85,B 0,C 180,E1 -5501.765,E2 -5501.765} C_VEL
LIN {X 0,Y 510.371,Z 665.466,A -85,B 0,C 180,E1 -5503.132,E2 -5503.132} C_VEL
LIN {X 0,Y 510.753,Z 655.092,A -85,B 0,C 180,E1 -5504.339,E2 -5504.339} C_VEL
LIN {X 0,Y 511.291,Z 643.519,A -85,B 0,C 180,E1 -5505.47,E2 -5505.47} C_VEL
LIN {X 0,Y 511.829,Z 630.219,A -85,B 0,C 180,E1 -5506.553,E2 -5506.553} C_VEL
LIN {X 0,Y 512.45,Z 616.61,A -85,B 0,C 180,E1 -5507.456,E2 -5507.456} C_VEL
LIN {X 0,Y 512.89,Z 602.527,A -85,B 0,C 180,E1 -5508.214,E2 -5508.214} C_VEL
LIN {X 0,Y 513.398,Z 587.343,A -85,B 0,C 180,E1 -5508.845,E2 -5508.845} C_VEL
LIN {X 0,Y 513.771,Z 571.963,A -85,B 0,C 180,E1 -5509.309,E2 -5509.309} C_VEL
LIN {X 0,Y 514.034,Z 555.289,A -85,B 0,C 180,E1 -5509.628,E2 -5509.628} C_VEL
LIN {X 0,Y 515.254,Z 414.35,A -85,B 0,C 180,E1 -5511.689,E2 -5511.689} C_VEL
LIN {X 0,Y 512.074,Z 397.932,A -85,B 0,C 180,E1 -5512.101,E2 -5512.101} C_VEL
LIN {X 0,Y 512.759,Z 380.16,A -85,B 0,C 180,E1 -5514.493,E2 -5514.493} C_VEL
LIN {X 0,Y 513.255,Z 367.601,A -85,B 0,C 180,E1 -5516.204,E2 -5516.204} C_VEL
LIN {X 0,Y 512.453,Z 362.578,A -85,B 0,C 180,E1 -5516.946,E2 -5516.946} C_VEL
LIN {X 0,Y 509.859,Z 351.603,A -85,B 0,C 180,E1 -5518.655,E2 -5518.655} C_VEL
LIN {X 0,Y 509.811,Z 351.606,A -85,B 0,C 180,E1 -5521.589,E2 -5521.589} C_VEL
LIN {X 0,Y 509.828,Z 351.605,A -85,B 0,C 180,E1 -5524.413,E2 -5524.413} C_VEL
LIN {X 0,Y 509.784,Z 351.606,A -85,B 0,C 180,E1 -5527.342,E2 -5527.342} C_VEL
LIN {X 0,Y 509.803,Z 351.608,A -85,B 0,C 180,E1 -5530.383,E2 -5530.383} C_VEL
LIN {X 0,Y 509.784,Z 351.604,A -85,B 0,C 180,E1 -5533.058,E2 -5533.058} C_VEL
LIN {X 0,Y 509.809,Z 351.604,A -85,B 0,C 180,E1 -5535.793,E2 -5535.793} C_VEL
LIN {X 0,Y 509.794,Z 351.606,A -85,B 0,C 180,E1 -5538.569,E2 -5538.569} C_VEL
LIN {X 0,Y 509.802,Z 351.604,A -85,B 0,C 180,E1 -5541.658,E2 -5541.658} C_VEL
LIN {X 0,Y 509.802,Z 351.604,A -85,B 0,C 180,E1 -5544.62,E2 -5544.62} C_VEL
LIN {X 0,Y 509.846,Z 351.597,A -85,B 0,C 180,E1 -5547.48,E2 -5547.48} C_VEL
LIN {X 0,Y 509.838,Z 351.604,A -85,B 0,C 180,E1 -5550.274,E2 -5550.274} C_VEL
LIN {X 0,Y 509.805,Z 351.601,A -85,B 0,C 180,E1 -5552.94,E2 -5552.94} C_VEL
LIN {X 0,Y 509.819,Z 351.601,A -85,B 0,C 180,E1 -5555.572,E2 -5555.572} C_VEL
LIN {X 0,Y 509.805,Z 351.61,A -85,B 0,C 180,E1 -5558.148,E2 -5558.148} C_VEL
LIN {X 0,Y 509.835,Z 351.599,A -85,B 0,C 180,E1 -5560.681,E2 -5560.681} C_VEL
LIN {X 0,Y 509.773,Z 351.605,A -85,B 0,C 180,E1 -5563.171,E2 -5563.171} C_VEL
LIN {X 0,Y 509.835,Z 351.601,A -85,B 0,C 180,E1 -5565.633,E2 -5565.633} C_VEL
LIN {X 0,Y 509.894,Z 351.59,A -85,B 0,C 180,E1 -5568.874,E2 -5568.874} C_VEL
LIN {X 0,Y 509.862,Z 351.603,A -85,B 0,C 180,E1 -5572.077,E2 -5572.077} C_VEL
LIN {X 0,Y 509.928,Z 351.589,A -85,B 0,C 180,E1 -5574.464,E2 -5574.464} C_VEL
LIN {X 0,Y 510.026,Z 351.577,A -85,B 0,C 180,E1 -5577.631,E2 -5577.631} C_VEL
LIN {X 0,Y 510.018,Z 351.584,A -85,B 0,C 180,E1 -5580,E2 -5580} C_VEL
LIN {X 0,Y 510.026,Z 351.577,A -85,B 0,C 180,E1 -5582.369,E2 -5582.369} C_VEL
LIN {X 0,Y 509.922,Z 351.589,A -85,B 0,C 180,E1 -5585.537,E2 -5585.537} C_VEL
LIN {X 0,Y 509.86,Z 351.603,A -85,B 0,C 180,E1 -5587.923,E2 -5587.923} C_VEL
LIN {X 0,Y 509.847,Z 351.596,A -85,B 0,C 180,E1 -5591.127,E2 -5591.127} C_VEL
LIN {X 0,Y 509.83,Z 351.601,A -85,B 0,C 180,E1 -5593.553,E2 -5593.553} C_VEL
LIN {X 0,Y 509.788,Z 351.612,A -85,B 0,C 180,E1 -5596.005,E2 -5596.005} C_VEL
LIN {X 0,Y 509.82,Z 351.601,A -85,B 0,C 180,E1 -5598.486,E2 -5598.486} C_VEL
LIN {X 0,Y 509.828,Z 351.598,A -85,B 0,C 180,E1 -5601.003,E2 -5601.003} C_VEL
LIN {X 0,Y 509.803,Z 351.605,A -85,B 0,C 180,E1 -5603.565,E2 -5603.565} C_VEL
LIN {X 0,Y 509.8,Z 351.605,A -85,B 0,C 180,E1 -5606.357,E2 -5606.357} C_VEL
LIN {X 0,Y 509.82,Z 351.599,A -85,B 0,C 180,E1 -5608.848,E2 -5608.848} C_VEL
LIN {X 0,Y 509.806,Z 351.606,A -85,B 0,C 180,E1 -5611.591,E2 -5611.591} C_VEL
LIN {X 0,Y 509.826,Z 351.6,A -85,B 0,C 180,E1 -5614.416,E2 -5614.416} C_VEL
LIN {X 0,Y 509.772,Z 351.607,A -85,B 0,C 180,E1 -5617.345,E2 -5617.345} C_VEL
LIN {X 0,Y 509.803,Z 351.603,A -85,B 0,C 180,E1 -5620.386,E2 -5620.386} C_VEL
LIN {X 0,Y 509.796,Z 351.607,A -85,B 0,C 180,E1 -5623.575,E2 -5623.575} C_VEL
LIN {X 0,Y 509.799,Z 351.603,A -85,B 0,C 180,E1 -5626.428,E2 -5626.428} C_VEL
LIN {X 0,Y 509.803,Z 351.604,A -85,B 0,C 180,E1 -5629.307,E2 -5629.307} C_VEL
LIN {X 0,Y 509.809,Z 351.61,A -85,B 0,C 180,E1 -5631.793,E2 -5631.793} C_VEL
LIN {X 0,Y 509.794,Z 351.609,A -85,B 0,C 180,E1 -5633.703,E2 -5633.703} C_VEL
LIN {X 0,Y 509.134,Z 351.687,A -85,B 0,C 180,E1 -5634.363,E2 -5634.363} C_VEL
LIN {X 0,Y 506.333,Z 352.038,A -85,B 0,C 180,E1 -5635.435,E2 -5635.435} C_VEL
LIN {X 0,Y 503.95,Z 352.333,A -85,B 0,C 180,E1 -5636.299,E2 -5636.299} C_VEL
LIN {X 0,Y 502.903,Z 352.461,A -85,B 0,C 180,E1 -5636.965,E2 -5636.965} C_VEL
LIN {X 0,Y 502.804,Z 352.474,A -85,B 0,C 180,E1 -5637.191,E2 -5637.191} C_VEL
LIN {X 0,Y 502.806,Z 352.478,A -85,B 0,C 180,E1 -5640.068,E2 -5640.068} C_VEL
LIN {X 0,Y 502.77,Z 352.482,A -85,B 0,C 180,E1 -5643.461,E2 -5643.461} C_VEL
LIN {X 0,Y 502.765,Z 352.482,A -85,B 0,C 180,E1 -5646.087,E2 -5646.087} C_VEL
LIN {X 0,Y 502.782,Z 352.476,A -85,B 0,C 180,E1 -5648.69,E2 -5648.69} C_VEL
LIN {X 0,Y 502.81,Z 352.475,A -85,B 0,C 180,E1 -5651.249,E2 -5651.249} C_VEL
LIN {X 0,Y 502.837,Z 352.469,A -85,B 0,C 180,E1 -5654.665,E2 -5654.665} C_VEL
LIN {X 0,Y 502.878,Z 352.468,A -85,B 0,C 180,E1 -5658.041,E2 -5658.041} C_VEL
LIN {X 0,Y 502.85,Z 352.47,A -85,B 0,C 180,E1 -5661.158,E2 -5661.158} C_VEL
LIN {X 0,Y 502.872,Z 352.472,A -85,B 0,C 180,E1 -5663.582,E2 -5663.582} C_VEL
LIN {X 0,Y 502.837,Z 352.469,A -85,B 0,C 180,E1 -5666.796,E2 -5666.796} C_VEL
LIN {X 0,Y 502.895,Z 352.463,A -85,B 0,C 180,E1 -5668.4,E2 -5668.4} C_VEL
LIN {X 0,Y 503.006,Z 352.452,A -85,B 0,C 180,E1 -5670.001,E2 -5670.001} C_VEL
LIN {X 0,Y 503.014,Z 352.448,A -85,B 0,C 180,E1 -5672.403,E2 -5672.403} C_VEL
LIN {X 0,Y 502.901,Z 352.47,A -85,B 0,C 180,E1 -5675.615,E2 -5675.615} C_VEL
LIN {X 0,Y 502.876,Z 352.468,A -85,B 0,C 180,E1 -5678.035,E2 -5678.035} C_VEL
LIN {X 0,Y 502.881,Z 352.468,A -85,B 0,C 180,E1 -5681.284,E2 -5681.284} C_VEL
LIN {X 0,Y 502.838,Z 352.469,A -85,B 0,C 180,E1 -5684.572,E2 -5684.572} C_VEL
LIN {X 0,Y 502.815,Z 352.474,A -85,B 0,C 180,E1 -5688.11,E2 -5688.11} C_VEL
LIN {X 0,Y 502.836,Z 352.469,A -85,B 0,C 180,E1 -5690.537,E2 -5690.537} C_VEL
LIN {X 0,Y 502.792,Z 352.477,A -85,B 0,C 180,E1 -5693.042,E2 -5693.042} C_VEL
LIN {X 0,Y 502.784,Z 352.483,A -85,B 0,C 180,E1 -5695.68,E2 -5695.68} C_VEL
LIN {X 0,Y 502.78,Z 352.477,A -85,B 0,C 180,E1 -5698.377,E2 -5698.377} C_VEL
LIN {X 0,Y 502.798,Z 352.477,A -85,B 0,C 180,E1 -5701.144,E2 -5701.144} C_VEL
LIN {X 0,Y 502.801,Z 352.476,A -85,B 0,C 180,E1 -5703.995,E2 -5703.995} C_VEL
LIN {X 0,Y 502.77,Z 352.485,A -85,B 0,C 180,E1 -5707.176,E2 -5707.176} C_VEL
LIN {X 0,Y 502.788,Z 352.481,A -85,B 0,C 180,E1 -5710.016,E2 -5710.016} C_VEL
LIN {X 0,Y 502.81,Z 352.477,A -85,B 0,C 180,E1 -5712.2,E2 -5712.2} C_VEL
LIN {X 0,Y 502.862,Z 352.617,A -85,B 0,C 180,E1 -5715.529,E2 -5715.529} C_VEL
LIN {X 0,Y 505.254,Z 363.916,A -85,B 0,C 180,E1 -5717.496,E2 -5717.496} C_VEL
LIN {X 0,Y 505.187,Z 371.331,A -85,B 0,C 180,E1 -5718.656,E2 -5718.656} C_VEL
LIN {X 0,Y 508.676,Z 386.853,A -85,B 0,C 180,E1 -5719.065,E2 -5719.065} C_VEL
LIN {X 0,Y 507.239,Z 536.585,A -85,B 0,C 180,E1 -5721.333,E2 -5721.333} C_VEL
LIN {X 0,Y 506.886,Z 552.127,A -85,B 0,C 180,E1 -5721.729,E2 -5721.729} C_VEL
LIN {X 0,Y 506.459,Z 567.057,A -85,B 0,C 180,E1 -5722.278,E2 -5722.278} C_VEL
LIN {X 0,Y 505.902,Z 582.029,A -85,B 0,C 180,E1 -5723.008,E2 -5723.008} C_VEL
LIN {X 0,Y 505.361,Z 595.69,A -85,B 0,C 180,E1 -5723.85,E2 -5723.85} C_VEL
LIN {X 0,Y 504.75,Z 608.61,A -85,B 0,C 180,E1 -5724.823,E2 -5724.823} C_VEL
LIN {X 0,Y 504.215,Z 620.181,A -85,B 0,C 180,E1 -5725.873,E2 -5725.873} C_VEL
LIN {X 0,Y 503.731,Z 630.945,A -85,B 0,C 180,E1 -5727.035,E2 -5727.035} C_VEL
LIN {X 0,Y 503.261,Z 641.704,A -85,B 0,C 180,E1 -5728.416,E2 -5728.416} C_VEL
LIN {X 0,Y 502.895,Z 650.647,A -85,B 0,C 180,E1 -5729.794,E2 -5729.794} C_VEL
LIN {X 0,Y 502.6,Z 658.026,A -85,B 0,C 180,E1 -5731.156,E2 -5731.156} C_VEL
LIN {X 0,Y 502.381,Z 664.198,A -85,B 0,C 180,E1 -5732.506,E2 -5732.506} C_VEL
LIN {X 0,Y 502.259,Z 669.515,A -85,B 0,C 180,E1 -5733.933,E2 -5733.933} C_VEL
LIN {X 0,Y 502.137,Z 674.024,A -85,B 0,C 180,E1 -5735.472,E2 -5735.472} C_VEL
LIN {X 0,Y 502.02,Z 678.239,A -85,B 0,C 180,E1 -5737.514,E2 -5737.514} C_VEL
LIN {X 0,Y 501.991,Z 679.739,A -85,B 0,C 180,E1 -5738.653,E2 -5738.653} C_VEL
LIN {X 0,Y 501.992,Z 680.894,A -85,B 0,C 180,E1 -5740.366,E2 -5740.366} C_VEL
LIN {X 0,Y 502.001,Z 680.74,A -85,B 0,C 180,E1 -5742.177,E2 -5742.177} C_VEL
LIN {X 0,Y 501.982,Z 679.42,A -85,B 0,C 180,E1 -5743.739,E2 -5743.739} C_VEL
LIN {X 0,Y 502.05,Z 676.819,A -85,B 0,C 180,E1 -5745.405,E2 -5745.405} C_VEL
LIN {X 0,Y 502.172,Z 672.892,A -85,B 0,C 180,E1 -5747.06,E2 -5747.06} C_VEL
LIN {X 0,Y 502.293,Z 667.665,A -85,B 0,C 180,E1 -5748.703,E2 -5748.703} C_VEL
LIN {X 0,Y 502.479,Z 660.97,A -85,B 0,C 180,E1 -5750.338,E2 -5750.338} C_VEL
LIN {X 0,Y 502.744,Z 653.766,A -85,B 0,C 180,E1 -5751.762,E2 -5751.762} C_VEL
LIN {X 0,Y 503.114,Z 644.712,A -85,B 0,C 180,E1 -5753.244,E2 -5753.244} C_VEL
LIN {X 0,Y 503.561,Z 634.783,A -85,B 0,C 180,E1 -5754.594,E2 -5754.594} C_VEL
LIN {X 0,Y 504.027,Z 624.21,A -85,B 0,C 180,E1 -5755.802,E2 -5755.802} C_VEL
LIN {X 0,Y 504.596,Z 611.567,A -85,B 0,C 180,E1 -5757.006,E2 -5757.006} C_VEL
LIN {X 0,Y 505.174,Z 598.842,A -85,B 0,C 180,E1 -5758.007,E2 -5758.007} C_VEL
LIN {X 0,Y 505.782,Z 584.834,A -85,B 0,C 180,E1 -5758.905,E2 -5758.905} C_VEL
LIN {X 0,Y 506.299,Z 570.526,A -85,B 0,C 180,E1 -5759.635,E2 -5759.635} C_VEL
LIN {X 0,Y 506.741,Z 556.178,A -85,B 0,C 180,E1 -5760.198,E2 -5760.198} C_VEL
LIN {X 0,Y 507.067,Z 541.369,A -85,B 0,C 180,E1 -5760.62,E2 -5760.62} C_VEL
LIN {X 0,Y 507.265,Z 523.458,A -85,B 0,C 180,E1 -5760.942,E2 -5760.942} C_VEL
LIN {X 0,Y 508.687,Z 389.71,A -85,B 0,C 180,E1 -5762.98,E2 -5762.98} C_VEL
LIN {X 0,Y 508.308,Z 385.062,A -85,B 0,C 180,E1 -5763.073,E2 -5763.073} C_VEL
LIN {X 0,Y 505.295,Z 371.952,A -85,B 0,C 180,E1 -5763.438,E2 -5763.438} C_VEL
LIN {X 0,Y 505.567,Z 364.842,A -85,B 0,C 180,E1 -5764.584,E2 -5764.584} C_VEL
LIN {X 0,Y 503.392,Z 354.614,A -85,B 0,C 180,E1 -5766.413,E2 -5766.413} C_VEL
LIN {X 0,Y 502.922,Z 352.467,A -85,B 0,C 180,E1 -5766.846,E2 -5766.846} C_VEL
LIN {X 0,Y 502.831,Z 352.476,A -85,B 0,C 180,E1 -5769.655,E2 -5769.655} C_VEL
LIN {X 0,Y 502.85,Z 352.473,A -85,B 0,C 180,E1 -5772.101,E2 -5772.101} C_VEL
LIN {X 0,Y 502.853,Z 352.471,A -85,B 0,C 180,E1 -5775.399,E2 -5775.399} C_VEL
LIN {X 0,Y 502.826,Z 352.477,A -85,B 0,C 180,E1 -5778.752,E2 -5778.752} C_VEL
LIN {X 0,Y 502.787,Z 352.477,A -85,B 0,C 180,E1 -5781.311,E2 -5781.311} C_VEL
LIN {X 0,Y 502.771,Z 352.483,A -85,B 0,C 180,E1 -5783.915,E2 -5783.915} C_VEL
LIN {X 0,Y 502.786,Z 352.482,A -85,B 0,C 180,E1 -5786.57,E2 -5786.57} C_VEL
LIN {X 0,Y 502.813,Z 352.479,A -85,B 0,C 180,E1 -5789.933,E2 -5789.933} C_VEL
LIN {X 0,Y 502.805,Z 352.475,A -85,B 0,C 180,E1 -5793.033,E2 -5793.033} C_VEL
LIN {X 0,Y 502.746,Z 352.488,A -85,B 0,C 180,E1 -5795.953,E2 -5795.953} C_VEL
LIN {X 0,Y 502.778,Z 352.478,A -85,B 0,C 180,E1 -5798.978,E2 -5798.978} C_VEL
LIN {X 0,Y 502.747,Z 352.488,A -85,B 0,C 180,E1 -5802.191,E2 -5802.191} C_VEL
LIN {X 0,Y 502.78,Z 352.479,A -85,B 0,C 180,E1 -5805.471,E2 -5805.471} C_VEL
LIN {X 0,Y 502.751,Z 352.481,A -85,B 0,C 180,E1 -5808.926,E2 -5808.926} C_VEL
LIN {X 0,Y 502.756,Z 352.488,A -85,B 0,C 180,E1 -5812.042,E2 -5812.042} C_VEL
LIN {X 0,Y 502.755,Z 352.484,A -85,B 0,C 180,E1 -5815.03,E2 -5815.03} C_VEL
LIN {X 0,Y 502.763,Z 352.491,A -85,B 0,C 180,E1 -5817.913,E2 -5817.913} C_VEL
LIN {X 0,Y 502.799,Z 352.482,A -85,B 0,C 180,E1 -5821.111,E2 -5821.111} C_VEL
LIN {X 0,Y 506.186,Z 367.024,A -85,B 0,C 180,E1 -5823.439,E2 -5823.439} C_VEL
LIN {X 0,Y 505.978,Z 376.735,A -85,B 0,C 180,E1 -5824.798,E2 -5824.798} C_VEL
LIN {X 0,Y 505.169,Z 397.105,A -85,B 0,C 180,E1 -5827.584,E2 -5827.584} C_VEL
LIN {X 0,Y 508.618,Z 415.382,A -85,B 0,C 180,E1 -5828.045,E2 -5828.045} C_VEL
LIN {X 0,Y 507.068,Z 564.517,A -85,B 0,C 180,E1 -5830.321,E2 -5830.321} C_VEL
LIN {X 0,Y 506.71,Z 579.984,A -85,B 0,C 180,E1 -5830.716,E2 -5830.716} C_VEL
LIN {X 0,Y 506.305,Z 594.497,A -85,B 0,C 180,E1 -5831.244,E2 -5831.244} C_VEL
LIN {X 0,Y 505.781,Z 608.035,A -85,B 0,C 180,E1 -5831.885,E2 -5831.885} C_VEL
LIN {X 0,Y 505.246,Z 621.789,A -85,B 0,C 180,E1 -5832.702,E2 -5832.702} C_VEL
LIN {X 0,Y 504.668,Z 634.437,A -85,B 0,C 180,E1 -5833.619,E2 -5833.619} C_VEL
LIN {X 0,Y 504.158,Z 646.188,A -85,B 0,C 180,E1 -5834.64,E2 -5834.64} C_VEL
LIN {X 0,Y 503.689,Z 656.197,A -85,B 0,C 180,E1 -5835.659,E2 -5835.659} C_VEL
LIN {X 0,Y 503.279,Z 666.438,A -85,B 0,C 180,E1 -5836.883,E2 -5836.883} C_VEL
LIN {X 0,Y 502.85,Z 675.746,A -85,B 0,C 180,E1 -5838.199,E2 -5838.199} C_VEL
LIN {X 0,Y 502.594,Z 684.724,A -85,B 0,C 180,E1 -5839.729,E2 -5839.729} C_VEL
LIN {X 0,Y 502.375,Z 691.562,A -85,B 0,C 180,E1 -5841.147,E2 -5841.147} C_VEL
LIN {X 0,Y 502.241,Z 697.888,A -85,B 0,C 180,E1 -5842.764,E2 -5842.764} C_VEL
LIN {X 0,Y 502.181,Z 702.773,A -85,B 0,C 180,E1 -5844.377,E2 -5844.377} C_VEL
LIN {X 0,Y 502.083,Z 706.351,A -85,B 0,C 180,E1 -5845.986,E2 -5845.986} C_VEL
LIN {X 0,Y 502.088,Z 708.707,A -85,B 0,C 180,E1 -5847.592,E2 -5847.592} C_VEL
LIN {X 0,Y 501.987,Z 709.892,A -85,B 0,C 180,E1 -5849.197,E2 -5849.197} C_VEL
LIN {X 0,Y 501.986,Z 709.897,A -85,B 0,C 180,E1 -5850.801,E2 -5850.801} C_VEL
LIN {X 0,Y 502.088,Z 708.724,A -85,B 0,C 180,E1 -5852.405,E2 -5852.405} C_VEL
LIN {X 0,Y 502.094,Z 706.387,A -85,B 0,C 180,E1 -5854.012,E2 -5854.012} C_VEL
LIN {X 0,Y 502.182,Z 702.836,A -85,B 0,C 180,E1 -5855.621,E2 -5855.621} C_VEL
LIN {X 0,Y 502.24,Z 697.976,A -85,B 0,C 180,E1 -5857.234,E2 -5857.234} C_VEL
LIN {X 0,Y 502.386,Z 691.676,A -85,B 0,C 180,E1 -5858.851,E2 -5858.851} C_VEL
LIN {X 0,Y 502.64,Z 683.757,A -85,B 0,C 180,E1 -5860.471,E2 -5860.471} C_VEL
LIN {X 0,Y 502.909,Z 675.723,A -85,B 0,C 180,E1 -5861.833,E2 -5861.833} C_VEL
LIN {X 0,Y 503.313,Z 666.712,A -85,B 0,C 180,E1 -5863.114,E2 -5863.114} C_VEL
LIN {X 0,Y 503.709,Z 656.558,A -85,B 0,C 180,E1 -5864.338,E2 -5864.338} C_VEL
LIN {X 0,Y 504.269,Z 645.089,A -85,B 0,C 180,E1 -5865.503,E2 -5865.503} C_VEL
LIN {X 0,Y 504.802,Z 632.411,A -85,B 0,C 180,E1 -5866.582,E2 -5866.582} C_VEL
LIN {X 0,Y 505.429,Z 619.327,A -85,B 0,C 180,E1 -5867.498,E2 -5867.498} C_VEL
LIN {X 0,Y 505.979,Z 604.975,A -85,B 0,C 180,E1 -5868.315,E2 -5868.315} C_VEL
LIN {X 0,Y 506.487,Z 591.04,A -85,B 0,C 180,E1 -5868.937,E2 -5868.937} C_VEL
LIN {X 0,Y 506.899,Z 575.445,A -85,B 0,C 180,E1 -5869.458,E2 -5869.458} C_VEL
LIN {X 0,Y 507.217,Z 560.936,A -85,B 0,C 180,E1 -5869.785,E2 -5869.785} C_VEL
LIN {X 0,Y 508.227,Z 457.628,A -85,B 0,C 180,E1 -5871.323,E2 -5871.323} C_VEL
LIN {X 0,Y 508.565,Z 414.767,A -85,B 0,C 180,E1 -5871.98,E2 -5871.98} C_VEL
LIN {X 0,Y 505.259,Z 397.761,A -85,B 0,C 180,E1 -5872.415,E2 -5872.415} C_VEL
LIN {X 0,Y 506.05,Z 378.417,A -85,B 0,C 180,E1 -5875.059,E2 -5875.059} C_VEL
LIN {X 0,Y 506.37,Z 367.658,A -85,B 0,C 180,E1 -5876.556,E2 -5876.556} C_VEL
LIN {X 0,Y 502.825,Z 352.478,A -85,B 0,C 180,E1 -5878.942,E2 -5878.942} C_VEL
LIN {X 0,Y 502.774,Z 352.484,A -85,B 0,C 180,E1 -5882.083,E2 -5882.083} C_VEL
LIN {X 0,Y 502.783,Z 352.479,A -85,B 0,C 180,E1 -5884.965,E2 -5884.965} C_VEL
LIN {X 0,Y 502.754,Z 352.486,A -85,B 0,C 180,E1 -5888.48,E2 -5888.48} C_VEL
LIN {X 0,Y 502.761,Z 352.479,A -85,B 0,C 180,E1 -5891.07,E2 -5891.07} C_VEL
LIN {X 0,Y 502.742,Z 352.481,A -85,B 0,C 180,E1 -5893.371,E2 -5893.371} C_VEL
LIN {X 0,Y 502.766,Z 352.48,A -85,B 0,C 180,E1 -5895.659,E2 -5895.659} C_VEL
LIN {X 0,Y 502.751,Z 352.48,A -85,B 0,C 180,E1 -5898.927,E2 -5898.927} C_VEL
LIN {X 0,Y 502.748,Z 352.488,A -85,B 0,C 180,E1 -5902.042,E2 -5902.042} C_VEL
LIN {X 0,Y 502.776,Z 352.477,A -85,B 0,C 180,E1 -5905.033,E2 -5905.033} C_VEL
LIN {X 0,Y 502.768,Z 352.483,A -85,B 0,C 180,E1 -5907.915,E2 -5907.915} C_VEL
LIN {X 0,Y 502.788,Z 352.477,A -85,B 0,C 180,E1 -5910.71,E2 -5910.71} C_VEL
LIN {X 0,Y 502.758,Z 352.48,A -85,B 0,C 180,E1 -5913.459,E2 -5913.459} C_VEL
LIN {X 0,Y 502.752,Z 352.489,A -85,B 0,C 180,E1 -5916.084,E2 -5916.084} C_VEL
LIN {X 0,Y 502.763,Z 352.48,A -85,B 0,C 180,E1 -5918.688,E2 -5918.688} C_VEL
LIN {X 0,Y 502.794,Z 352.475,A -85,B 0,C 180,E1 -5921.247,E2 -5921.247} C_VEL
LIN {X 0,Y 502.819,Z 352.473,A -85,B 0,C 180,E1 -5924.664,E2 -5924.664} C_VEL
LIN {X 0,Y 502.861,Z 352.475,A -85,B 0,C 180,E1 -5928.039,E2 -5928.039} C_VEL
LIN {X 0,Y 502.834,Z 352.47,A -85,B 0,C 180,E1 -5931.156,E2 -5931.156} C_VEL
LIN {X 0,Y 502.861,Z 352.469,A -85,B 0,C 180,E1 -5933.581,E2 -5933.581} C_VEL
LIN {X 0,Y 502.815,Z 352.472,A -85,B 0,C 180,E1 -5936.795,E2 -5936.795} C_VEL
LIN {X 0,Y 502.876,Z 352.468,A -85,B 0,C 180,E1 -5938.399,E2 -5938.399} C_VEL
LIN {X 0,Y 502.987,Z 352.46,A -85,B 0,C 180,E1 -5940,E2 -5940} C_VEL
LIN {X 0,Y 502.993,Z 352.453,A -85,B 0,C 180,E1 -5942.403,E2 -5942.403} C_VEL
LIN {X 0,Y 502.879,Z 352.468,A -85,B 0,C 180,E1 -5945.614,E2 -5945.614} C_VEL
LIN {X 0,Y 502.833,Z 352.478,A -85,B 0,C 180,E1 -5948.035,E2 -5948.035} C_VEL
LIN {X 0,Y 502.822,Z 352.472,A -85,B 0,C 180,E1 -5951.285,E2 -5951.285} C_VEL
LIN {X 0,Y 502.814,Z 352.473,A -85,B 0,C 180,E1 -5954.572,E2 -5954.572} C_VEL
LIN {X 0,Y 502.794,Z 352.481,A -85,B 0,C 180,E1 -5958.11,E2 -5958.11} C_VEL
LIN {X 0,Y 502.816,Z 352.473,A -85,B 0,C 180,E1 -5960.537,E2 -5960.537} C_VEL
LIN {X 0,Y 502.772,Z 352.477,A -85,B 0,C 180,E1 -5963.042,E2 -5963.042} C_VEL
LIN {X 0,Y 502.761,Z 352.484,A -85,B 0,C 180,E1 -5965.68,E2 -5965.68} C_VEL
LIN {X 0,Y 502.756,Z 352.482,A -85,B 0,C 180,E1 -5968.378,E2 -5968.378} C_VEL
LIN {X 0,Y 502.779,Z 352.477,A -85,B 0,C 180,E1 -5971.145,E2 -5971.145} C_VEL
LIN {X 0,Y 502.781,Z 352.483,A -85,B 0,C 180,E1 -5973.996,E2 -5973.996} C_VEL
LIN {X 0,Y 502.726,Z 352.484,A -85,B 0,C 180,E1 -5977.173,E2 -5977.173} C_VEL
LIN {X 0,Y 502.76,Z 352.485,A -85,B 0,C 180,E1 -5980.018,E2 -5980.018} C_VEL
LIN {X 0,Y 502.737,Z 352.483,A -85,B 0,C 180,E1 -5983.236,E2 -5983.236} C_VEL
LIN {X 0,Y 502.77,Z 352.484,A -85,B 0,C 180,E1 -5985.661,E2 -5985.661} C_VEL
LIN {X 0,Y 502.761,Z 352.479,A -85,B 0,C 180,E1 -5989.013,E2 -5989.013} C_VEL
LIN {X 0,Y 502.758,Z 352.484,A -85,B 0,C 180,E1 -5992.045,E2 -5992.045} C_VEL
LIN {X 0,Y 502.785,Z 352.476,A -85,B 0,C 180,E1 -5995.035,E2 -5995.035} C_VEL
LIN {X 0,Y 502.804,Z 352.474,A -85,B 0,C 180,E1 -5997.191,E2 -5997.191} C_VEL
LIN {X 0,Y 502.103,Z 352.569,A -85,B 0,C 180,E1 -5997.859,E2 -5997.859} C_VEL
LIN {X 0,Y 499.242,Z 352.919,A -85,B 0,C 180,E1 -5998.945,E2 -5998.945} C_VEL
LIN {X 0,Y 496.841,Z 353.225,A -85,B 0,C 180,E1 -5999.82,E2 -5999.82} C_VEL
LIN {X 0,Y 495.807,Z 353.346,A -85,B 0,C 180,E1 -6000.495,E2 -6000.495} C_VEL
LIN {X 0,Y 495.72,Z 353.356,A -85,B 0,C 180,E1 -6000.724,E2 -6000.724} C_VEL
LIN {X 0,Y 495.714,Z 353.363,A -85,B 0,C 180,E1 -6003.929,E2 -6003.929} C_VEL
LIN {X 0,Y 495.757,Z 353.353,A -85,B 0,C 180,E1 -6007.141,E2 -6007.141} C_VEL
LIN {X 0,Y 495.767,Z 353.354,A -85,B 0,C 180,E1 -6010.111,E2 -6010.111} C_VEL
LIN {X 0,Y 495.741,Z 353.353,A -85,B 0,C 180,E1 -6012.681,E2 -6012.681} C_VEL
LIN {X 0,Y 495.781,Z 353.35,A -85,B 0,C 180,E1 -6015.218,E2 -6015.218} C_VEL
LIN {X 0,Y 495.852,Z 353.34,A -85,B 0,C 180,E1 -6018.556,E2 -6018.556} C_VEL
LIN {X 0,Y 495.815,Z 353.35,A -85,B 0,C 180,E1 -6021.852,E2 -6021.852} C_VEL
LIN {X 0,Y 495.857,Z 353.34,A -85,B 0,C 180,E1 -6024.307,E2 -6024.307} C_VEL
LIN {X 0,Y 495.979,Z 353.331,A -85,B 0,C 180,E1 -6027.565,E2 -6027.565} C_VEL
LIN {X 0,Y 495.975,Z 353.328,A -85,B 0,C 180,E1 -6030.001,E2 -6030.001} C_VEL
LIN {X 0,Y 495.98,Z 353.324,A -85,B 0,C 180,E1 -6032.438,E2 -6032.438} C_VEL
LIN {X 0,Y 495.859,Z 353.347,A -85,B 0,C 180,E1 -6035.695,E2 -6035.695} C_VEL
LIN {X 0,Y 495.835,Z 353.344,A -85,B 0,C 180,E1 -6038.15,E2 -6038.15} C_VEL
LIN {X 0,Y 495.856,Z 353.345,A -85,B 0,C 180,E1 -6041.446,E2 -6041.446} C_VEL
LIN {X 0,Y 495.787,Z 353.348,A -85,B 0,C 180,E1 -6044.784,E2 -6044.784} C_VEL
LIN {X 0,Y 495.778,Z 353.35,A -85,B 0,C 180,E1 -6048.235,E2 -6048.235} C_VEL
LIN {X 0,Y 495.781,Z 353.349,A -85,B 0,C 180,E1 -6050.757,E2 -6050.757} C_VEL
LIN {X 0,Y 495.745,Z 353.359,A -85,B 0,C 180,E1 -6053.388,E2 -6053.388} C_VEL
LIN {X 0,Y 495.745,Z 353.353,A -85,B 0,C 180,E1 -6056.73,E2 -6056.73} C_VEL
LIN {X 0,Y 495.764,Z 353.356,A -85,B 0,C 180,E1 -6059.748,E2 -6059.748} C_VEL
LIN {X 0,Y 495.774,Z 353.349,A -85,B 0,C 180,E1 -6062.595,E2 -6062.595} C_VEL
LIN {X 0,Y 495.75,Z 353.361,A -85,B 0,C 180,E1 -6065.539,E2 -6065.539} C_VEL
LIN {X 0,Y 495.766,Z 353.353,A -85,B 0,C 180,E1 -6068.768,E2 -6068.768} C_VEL
LIN {X 0,Y 495.756,Z 353.359,A -85,B 0,C 180,E1 -6071.782,E2 -6071.782} C_VEL
LIN {X 0,Y 495.776,Z 353.374,A -85,B 0,C 180,E1 -6075.245,E2 -6075.245} C_VEL
LIN {X 0,Y 498.397,Z 365.589,A -85,B 0,C 180,E1 -6077.401,E2 -6077.401} C_VEL
LIN {X 0,Y 498.343,Z 371.376,A -85,B 0,C 180,E1 -6078.333,E2 -6078.333} C_VEL
LIN {X 0,Y 502.12,Z 388.729,A -85,B 0,C 180,E1 -6078.794,E2 -6078.794} C_VEL
LIN {X 0,Y 500.51,Z 537.232,A -85,B 0,C 180,E1 -6081.086,E2 -6081.086} C_VEL
LIN {X 0,Y 500.12,Z 553.01,A -85,B 0,C 180,E1 -6081.502,E2 -6081.502} C_VEL
LIN {X 0,Y 499.719,Z 566.139,A -85,B 0,C 180,E1 -6081.987,E2 -6081.987} C_VEL
LIN {X 0,Y 499.162,Z 580.482,A -85,B 0,C 180,E1 -6082.678,E2 -6082.678} C_VEL
LIN {X 0,Y 498.58,Z 594.732,A -85,B 0,C 180,E1 -6083.549,E2 -6083.549} C_VEL
LIN {X 0,Y 497.919,Z 607.616,A -85,B 0,C 180,E1 -6084.516,E2 -6084.516} C_VEL
LIN {X 0,Y 497.38,Z 619.387,A -85,B 0,C 180,E1 -6085.583,E2 -6085.583} C_VEL
LIN {X 0,Y 496.804,Z 630.453,A -85,B 0,C 180,E1 -6086.775,E2 -6086.775} C_VEL
LIN {X 0,Y 496.31,Z 640.637,A -85,B 0,C 180,E1 -6088.078,E2 -6088.078} C_VEL
LIN {X 0,Y 495.944,Z 648.894,A -85,B 0,C 180,E1 -6089.326,E2 -6089.326} C_VEL
LIN {X 0,Y 495.617,Z 656.659,A -85,B 0,C 180,E1 -6090.71,E2 -6090.71} C_VEL
LIN {X 0,Y 495.392,Z 663.082,A -85,B 0,C 180,E1 -6092.085,E2 -6092.085} C_VEL
LIN {X 0,Y 495.235,Z 668.142,A -85,B 0,C 180,E1 -6093.388,E2 -6093.388} C_VEL
LIN {X 0,Y 495.091,Z 672.625,A -85,B 0,C 180,E1 -6094.795,E2 -6094.795} C_VEL
LIN {X 0,Y 494.978,Z 676.872,A -85,B 0,C 180,E1 -6096.574,E2 -6096.574} C_VEL
LIN {X 0,Y 494.894,Z 679.622,A -85,B 0,C 180,E1 -6098.332,E2 -6098.332} C_VEL
LIN {X 0,Y 494.891,Z 681.029,A -85,B 0,C 180,E1 -6100.072,E2 -6100.072} C_VEL
LIN {X 0,Y 494.893,Z 681.102,A -85,B 0,C 180,E1 -6101.794,E2 -6101.794} C_VEL
LIN {X 0,Y 494.885,Z 679.934,A -85,B 0,C 180,E1 -6103.499,E2 -6103.499} C_VEL
LIN {X 0,Y 494.951,Z 677.503,A -85,B 0,C 180,E1 -6105.191,E2 -6105.191} C_VEL
LIN {X 0,Y 495.058,Z 673.802,A -85,B 0,C 180,E1 -6106.871,E2 -6106.871} C_VEL
LIN {X 0,Y 495.199,Z 668.778,A -85,B 0,C 180,E1 -6108.539,E2 -6108.539} C_VEL
LIN {X 0,Y 495.394,Z 662.319,A -85,B 0,C 180,E1 -6110.198,E2 -6110.198} C_VEL
LIN {X 0,Y 495.707,Z 654.248,A -85,B 0,C 180,E1 -6111.849,E2 -6111.849} C_VEL
LIN {X 0,Y 496.079,Z 646.116,A -85,B 0,C 180,E1 -6113.218,E2 -6113.218} C_VEL
LIN {X 0,Y 496.485,Z 636.979,A -85,B 0,C 180,E1 -6114.517,E2 -6114.517} C_VEL
LIN {X 0,Y 496.994,Z 626.766,A -85,B 0,C 180,E1 -6115.742,E2 -6115.742} C_VEL
LIN {X 0,Y 497.565,Z 614.582,A -85,B 0,C 180,E1 -6116.964,E2 -6116.964} C_VEL
LIN {X 0,Y 498.229,Z 602.383,A -85,B 0,C 180,E1 -6117.979,E2 -6117.979} C_VEL
LIN {X 0,Y 498.794,Z 589.165,A -85,B 0,C 180,E1 -6118.89,E2 -6118.89} C_VEL
LIN {X 0,Y 499.39,Z 574.309,A -85,B 0,C 180,E1 -6119.709,E2 -6119.709} C_VEL
LIN {X 0,Y 499.869,Z 559.115,A -85,B 0,C 180,E1 -6120.352,E2 -6120.352} C_VEL
LIN {X 0,Y 500.307,Z 543.363,A -85,B 0,C 180,E1 -6120.83,E2 -6120.83} C_VEL
LIN {X 0,Y 500.492,Z 528.153,A -85,B 0,C 180,E1 -6121.131,E2 -6121.131} C_VEL
LIN {X 0,Y 502.059,Z 395.721,A -85,B 0,C 180,E1 -6123.189,E2 -6123.189} C_VEL
LIN {X 0,Y 501.978,Z 387.324,A -85,B 0,C 180,E1 -6123.335,E2 -6123.335} C_VEL
LIN {X 0,Y 498.553,Z 372.245,A -85,B 0,C 180,E1 -6123.768,E2 -6123.768} C_VEL
LIN {X 0,Y 498.773,Z 366.874,A -85,B 0,C 180,E1 -6124.647,E2 -6124.647} C_VEL
LIN {X 0,Y 496.937,Z 357.791,A -85,B 0,C 180,E1 -6126.292,E2 -6126.292} C_VEL
LIN {X 0,Y 495.902,Z 353.341,A -85,B 0,C 180,E1 -6127.155,E2 -6127.155} C_VEL
LIN {X 0,Y 495.791,Z 353.354,A -85,B 0,C 180,E1 -6129.794,E2 -6129.794} C_VEL
LIN {X 0,Y 495.793,Z 353.355,A -85,B 0,C 180,E1 -6132.276,E2 -6132.276} C_VEL
LIN {X 0,Y 495.828,Z 353.347,A -85,B 0,C 180,E1 -6135.451,E2 -6135.451} C_VEL
LIN {X 0,Y 495.782,Z 353.352,A -85,B 0,C 180,E1 -6139.028,E2 -6139.028} C_VEL
LIN {X 0,Y 495.746,Z 353.355,A -85,B 0,C 180,E1 -6141.629,E2 -6141.629} C_VEL
LIN {X 0,Y 495.717,Z 353.364,A -85,B 0,C 180,E1 -6144.277,E2 -6144.277} C_VEL
LIN {X 0,Y 495.732,Z 353.358,A -85,B 0,C 180,E1 -6146.979,E2 -6146.979} C_VEL
LIN {X 0,Y 495.76,Z 353.358,A -85,B 0,C 180,E1 -6150.145,E2 -6150.145} C_VEL
LIN {X 0,Y 495.754,Z 353.353,A -85,B 0,C 180,E1 -6153.236,E2 -6153.236} C_VEL
LIN {X 0,Y 495.689,Z 353.367,A -85,B 0,C 180,E1 -6156.082,E2 -6156.082} C_VEL
LIN {X 0,Y 495.737,Z 353.356,A -85,B 0,C 180,E1 -6158.763,E2 -6158.763} C_VEL
LIN {X 0,Y 495.703,Z 353.365,A -85,B 0,C 180,E1 -6161.786,E2 -6161.786} C_VEL
LIN {X 0,Y 495.733,Z 353.355,A -85,B 0,C 180,E1 -6165.141,E2 -6165.141} C_VEL
LIN {X 0,Y 495.702,Z 353.364,A -85,B 0,C 180,E1 -6168.212,E2 -6168.212} C_VEL
LIN {X 0,Y 495.715,Z 353.361,A -85,B 0,C 180,E1 -6171.404,E2 -6171.404} C_VEL
LIN {X 0,Y 495.717,Z 353.363,A -85,B 0,C 180,E1 -6174.459,E2 -6174.459} C_VEL
LIN {X 0,Y 495.728,Z 353.365,A -85,B 0,C 180,E1 -6177.402,E2 -6177.402} C_VEL
LIN {X 0,Y 495.755,Z 353.36,A -85,B 0,C 180,E1 -6180.719,E2 -6180.719} C_VEL
LIN {X 0,Y 495.768,Z 353.511,A -85,B 0,C 180,E1 -6180.836,E2 -6180.836} C_VEL
LIN {X 0,Y 499.233,Z 368.212,A -85,B 0,C 180,E1 -6183.224,E2 -6183.224} C_VEL
LIN {X 0,Y 499.438,Z 372.869,A -85,B 0,C 180,E1 -6183.911,E2 -6183.911} C_VEL
LIN {X 0,Y 498.353,Z 396.336,A -85,B 0,C 180,E1 -6187.181,E2 -6187.181} C_VEL
LIN {X 0,Y 498.392,Z 397.285,A -85,B 0,C 180,E1 -6187.264,E2 -6187.264} C_VEL
LIN {X 0,Y 502.043,Z 416.862,A -85,B 0,C 180,E1 -6187.769,E2 -6187.769} C_VEL
LIN {X 0,Y 500.34,Z 563.75,A -85,B 0,C 180,E1 -6190.057,E2 -6190.057} C_VEL
LIN {X 0,Y 499.93,Z 579.689,A -85,B 0,C 180,E1 -6190.467,E2 -6190.467} C_VEL
LIN {X 0,Y 499.47,Z 594.904,A -85,B 0,C 180,E1 -6191.033,E2 -6191.033} C_VEL
LIN {X 0,Y 498.878,Z 609.251,A -85,B 0,C 180,E1 -6191.732,E2 -6191.732} C_VEL
LIN {X 0,Y 498.319,Z 622.757,A -85,B 0,C 180,E1 -6192.56,E2 -6192.56} C_VEL
LIN {X 0,Y 497.727,Z 635.208,A -85,B 0,C 180,E1 -6193.49,E2 -6193.49} C_VEL
LIN {X 0,Y 497.103,Z 647.887,A -85,B 0,C 180,E1 -6194.627,E2 -6194.627} C_VEL
LIN {X 0,Y 496.588,Z 659.407,A -85,B 0,C 180,E1 -6195.868,E2 -6195.868} C_VEL
LIN {X 0,Y 496.065,Z 670.59,A -85,B 0,C 180,E1 -6197.314,E2 -6197.314} C_VEL
LIN {X 0,Y 495.691,Z 679.837,A -85,B 0,C 180,E1 -6198.757,E2 -6198.757} C_VEL
LIN {X 0,Y 495.387,Z 687.494,A -85,B 0,C 180,E1 -6200.197,E2 -6200.197} C_VEL
LIN {X 0,Y 495.224,Z 694.641,A -85,B 0,C 180,E1 -6201.84,E2 -6201.84} C_VEL
LIN {X 0,Y 495.086,Z 700.494,A -85,B 0,C 180,E1 -6203.557,E2 -6203.557} C_VEL
LIN {X 0,Y 495.003,Z 704.485,A -85,B 0,C 180,E1 -6205.112,E2 -6205.112} C_VEL
LIN {X 0,Y 495.025,Z 707.459,A -85,B 0,C 180,E1 -6206.743,E2 -6206.743} C_VEL
LIN {X 0,Y 494.96,Z 709.234,A -85,B 0,C 180,E1 -6208.371,E2 -6208.371} C_VEL
LIN {X 0,Y 494.895,Z 709.846,A -85,B 0,C 180,E1 -6209.999,E2 -6209.999} C_VEL
LIN {X 0,Y 494.959,Z 709.25,A -85,B 0,C 180,E1 -6211.626,E2 -6211.626} C_VEL
LIN {X 0,Y 495.026,Z 707.496,A -85,B 0,C 180,E1 -6213.254,E2 -6213.254} C_VEL
LIN {X 0,Y 495.003,Z 704.551,A -85,B 0,C 180,E1 -6214.886,E2 -6214.886} C_VEL
LIN {X 0,Y 495.16,Z 700.35,A -85,B 0,C 180,E1 -6216.519,E2 -6216.519} C_VEL
LIN {X 0,Y 495.227,Z 694.771,A -85,B 0,C 180,E1 -6218.157,E2 -6218.157} C_VEL
LIN {X 0,Y 495.388,Z 687.667,A -85,B 0,C 180,E1 -6219.801,E2 -6219.801} C_VEL
LIN {X 0,Y 495.703,Z 680.065,A -85,B 0,C 180,E1 -6221.24,E2 -6221.24} C_VEL
LIN {X 0,Y 496.065,Z 670.895,A -85,B 0,C 180,E1 -6222.684,E2 -6222.684} C_VEL
LIN {X 0,Y 496.597,Z 659.816,A -85,B 0,C 180,E1 -6224.129,E2 -6224.129} C_VEL
LIN {X 0,Y 497.158,Z 648.424,A -85,B 0,C 180,E1 -6225.369,E2 -6225.369} C_VEL
LIN {X 0,Y 497.774,Z 635.9,A -85,B 0,C 180,E1 -6226.506,E2 -6226.506} C_VEL
LIN {X 0,Y 498.361,Z 623.58,A -85,B 0,C 180,E1 -6227.436,E2 -6227.436} C_VEL
LIN {X 0,Y 498.964,Z 610.274,A -85,B 0,C 180,E1 -6228.262,E2 -6228.262} C_VEL
LIN {X 0,Y 499.555,Z 596.123,A -85,B 0,C 180,E1 -6228.966,E2 -6228.966} C_VEL
LIN {X 0,Y 500.027,Z 580.774,A -85,B 0,C 180,E1 -6229.549,E2 -6229.549} C_VEL
LIN {X 0,Y 500.413,Z 566.2,A -85,B 0,C 180,E1 -6229.937,E2 -6229.937} C_VEL
LIN {X 0,Y 500.732,Z 539.306,A -85,B 0,C 180,E1 -6230.379,E2 -6230.379} C_VEL
LIN {X 0,Y 502.027,Z 416.184,A -85,B 0,C 180,E1 -6232.256,E2 -6232.256} C_VEL
LIN {X 0,Y 498.418,Z 397.588,A -85,B 0,C 180,E1 -6232.74,E2 -6232.74} C_VEL
LIN {X 0,Y 499.477,Z 375.1,A -85,B 0,C 180,E1 -6235.859,E2 -6235.859} C_VEL
LIN {X 0,Y 499.439,Z 368.819,A -85,B 0,C 180,E1 -6236.761,E2 -6236.761} C_VEL
LIN {X 0,Y 495.766,Z 353.357,A -85,B 0,C 180,E1 -6239.249,E2 -6239.249} C_VEL
LIN {X 0,Y 495.758,Z 353.358,A -85,B 0,C 180,E1 -6242.593,E2 -6242.593} C_VEL
LIN {X 0,Y 495.733,Z 353.357,A -85,B 0,C 180,E1 -6245.537,E2 -6245.537} C_VEL
LIN {X 0,Y 495.73,Z 353.358,A -85,B 0,C 180,E1 -6248.764,E2 -6248.764} C_VEL
LIN {X 0,Y 495.732,Z 353.357,A -85,B 0,C 180,E1 -6251.781,E2 -6251.781} C_VEL
LIN {X 0,Y 495.725,Z 353.355,A -85,B 0,C 180,E1 -6255.14,E2 -6255.14} C_VEL
LIN {X 0,Y 495.711,Z 353.365,A -85,B 0,C 180,E1 -6258.214,E2 -6258.214} C_VEL
LIN {X 0,Y 495.727,Z 353.355,A -85,B 0,C 180,E1 -6261.234,E2 -6261.234} C_VEL
LIN {X 0,Y 495.722,Z 353.36,A -85,B 0,C 180,E1 -6264.46,E2 -6264.46} C_VEL
LIN {X 0,Y 495.753,Z 353.352,A -85,B 0,C 180,E1 -6267.405,E2 -6267.405} C_VEL
LIN {X 0,Y 495.742,Z 353.36,A -85,B 0,C 180,E1 -6270.252,E2 -6270.252} C_VEL
LIN {X 0,Y 495.723,Z 353.356,A -85,B 0,C 180,E1 -6273.27,E2 -6273.27} C_VEL
LIN {X 0,Y 495.723,Z 353.358,A -85,B 0,C 180,E1 -6276.612,E2 -6276.612} C_VEL
LIN {X 0,Y 495.764,Z 353.351,A -85,B 0,C 180,E1 -6279.324,E2 -6279.324} C_VEL
LIN {X 0,Y 495.764,Z 353.356,A -85,B 0,C 180,E1 -6281.828,E2 -6281.828} C_VEL
LIN {X 0,Y 495.763,Z 353.351,A -85,B 0,C 180,E1 -6285.217,E2 -6285.217} C_VEL
LIN {X 0,Y 495.834,Z 353.344,A -85,B 0,C 180,E1 -6288.555,E2 -6288.555} C_VEL
LIN {X 0,Y 495.798,Z 353.352,A -85,B 0,C 180,E1 -6291.851,E2 -6291.851} C_VEL
LIN {X 0,Y 495.843,Z 353.345,A -85,B 0,C 180,E1 -6294.306,E2 -6294.306} C_VEL
LIN {X 0,Y 495.96,Z 353.329,A -85,B 0,C 180,E1 -6297.564,E2 -6297.564} C_VEL
LIN {X 0,Y 495.956,Z 353.336,A -85,B 0,C 180,E1 -6300,E2 -6300} C_VEL
LIN {X 0,Y 495.959,Z 353.329,A -85,B 0,C 180,E1 -6302.437,E2 -6302.437} C_VEL
LIN {X 0,Y 495.837,Z 353.346,A -85,B 0,C 180,E1 -6305.694,E2 -6305.694} C_VEL
LIN {X 0,Y 495.797,Z 353.353,A -85,B 0,C 180,E1 -6308.149,E2 -6308.149} C_VEL
LIN {X 0,Y 495.806,Z 353.347,A -85,B 0,C 180,E1 -6311.447,E2 -6311.447} C_VEL
LIN {X 0,Y 495.764,Z 353.351,A -85,B 0,C 180,E1 -6314.784,E2 -6314.784} C_VEL
LIN {X 0,Y 495.757,Z 353.356,A -85,B 0,C 180,E1 -6318.235,E2 -6318.235} C_VEL
LIN {X 0,Y 495.76,Z 353.351,A -85,B 0,C 180,E1 -6320.757,E2 -6320.757} C_VEL
LIN {X 0,Y 495.724,Z 353.357,A -85,B 0,C 180,E1 -6323.389,E2 -6323.389} C_VEL
LIN {X 0,Y 495.724,Z 353.355,A -85,B 0,C 180,E1 -6326.73,E2 -6326.73} C_VEL
LIN {X 0,Y 495.744,Z 353.36,A -85,B 0,C 180,E1 -6329.748,E2 -6329.748} C_VEL
LIN {X 0,Y 495.755,Z 353.352,A -85,B 0,C 180,E1 -6332.596,E2 -6332.596} C_VEL
LIN {X 0,Y 495.724,Z 353.359,A -85,B 0,C 180,E1 -6335.54,E2 -6335.54} C_VEL
LIN {X 0,Y 495.729,Z 353.355,A -85,B 0,C 180,E1 -6338.766,E2 -6338.766} C_VEL
LIN {X 0,Y 495.713,Z 353.365,A -85,B 0,C 180,E1 -6341.786,E2 -6341.786} C_VEL
LIN {X 0,Y 495.728,Z 353.356,A -85,B 0,C 180,E1 -6345.142,E2 -6345.142} C_VEL
LIN {X 0,Y 495.717,Z 353.359,A -85,B 0,C 180,E1 -6348.217,E2 -6348.217} C_VEL
LIN {X 0,Y 495.733,Z 353.356,A -85,B 0,C 180,E1 -6351.237,E2 -6351.237} C_VEL
LIN {X 0,Y 495.735,Z 353.355,A -85,B 0,C 180,E1 -6354.463,E2 -6354.463} C_VEL
LIN {X 0,Y 495.761,Z 353.354,A -85,B 0,C 180,E1 -6357.407,E2 -6357.407} C_VEL
LIN {X 0,Y 495.752,Z 353.354,A -85,B 0,C 180,E1 -6360.255,E2 -6360.255} C_VEL
LIN {X 0,Y 495.72,Z 353.356,A -85,B 0,C 180,E1 -6360.724,E2 -6360.724} C_VEL
LIN {X 0,Y 495.039,Z 353.446,A -85,B 0,C 180,E1 -6361.403,E2 -6361.403} C_VEL
LIN {X 0,Y 492.165,Z 353.799,A -85,B 0,C 180,E1 -6362.505,E2 -6362.505} C_VEL
LIN {X 0,Y 489.751,Z 354.103,A -85,B 0,C 180,E1 -6363.393,E2 -6363.393} C_VEL
LIN {X 0,Y 488.729,Z 354.231,A -85,B 0,C 180,E1 -6364.079,E2 -6364.079} C_VEL
LIN {X 0,Y 488.654,Z 354.237,A -85,B 0,C 180,E1 -6364.311,E2 -6364.311} C_VEL
LIN {X 0,Y 488.719,Z 354.229,A -85,B 0,C 180,E1 -6367.155,E2 -6367.155} C_VEL
LIN {X 0,Y 488.722,Z 354.235,A -85,B 0,C 180,E1 -6369.812,E2 -6369.812} C_VEL
LIN {X 0,Y 488.699,Z 354.231,A -85,B 0,C 180,E1 -6372.424,E2 -6372.424} C_VEL
LIN {X 0,Y 488.756,Z 354.224,A -85,B 0,C 180,E1 -6375.001,E2 -6375.001} C_VEL
LIN {X 0,Y 488.806,Z 354.218,A -85,B 0,C 180,E1 -6378.389,E2 -6378.389} C_VEL
LIN {X 0,Y 488.763,Z 354.231,A -85,B 0,C 180,E1 -6381.734,E2 -6381.734} C_VEL
LIN {X 0,Y 488.816,Z 354.218,A -85,B 0,C 180,E1 -6384.225,E2 -6384.225} C_VEL
LIN {X 0,Y 488.945,Z 354.207,A -85,B 0,C 180,E1 -6387.53,E2 -6387.53} C_VEL
LIN {X 0,Y 488.945,Z 354.204,A -85,B 0,C 180,E1 -6390.001,E2 -6390.001} C_VEL
LIN {X 0,Y 488.947,Z 354.2,A -85,B 0,C 180,E1 -6392.473,E2 -6392.473} C_VEL
LIN {X 0,Y 488.819,Z 354.222,A -85,B 0,C 180,E1 -6395.777,E2 -6395.777} C_VEL
LIN {X 0,Y 488.784,Z 354.221,A -85,B 0,C 180,E1 -6398.268,E2 -6398.268} C_VEL
LIN {X 0,Y 488.81,Z 354.226,A -85,B 0,C 180,E1 -6401.613,E2 -6401.613} C_VEL
LIN {X 0,Y 488.756,Z 354.225,A -85,B 0,C 180,E1 -6405.002,E2 -6405.002} C_VEL
LIN {X 0,Y 488.75,Z 354.224,A -85,B 0,C 180,E1 -6408.443,E2 -6408.443} C_VEL
LIN {X 0,Y 488.713,Z 354.231,A -85,B 0,C 180,E1 -6411.072,E2 -6411.072} C_VEL
LIN {X 0,Y 488.675,Z 354.24,A -85,B 0,C 180,E1 -6413.747,E2 -6413.747} C_VEL
LIN {X 0,Y 488.704,Z 354.231,A -85,B 0,C 180,E1 -6416.922,E2 -6416.922} C_VEL
LIN {X 0,Y 488.724,Z 354.228,A -85,B 0,C 180,E1 -6420.22,E2 -6420.22} C_VEL
LIN {X 0,Y 488.738,Z 354.234,A -85,B 0,C 180,E1 -6423.484,E2 -6423.484} C_VEL
LIN {X 0,Y 488.679,Z 354.237,A -85,B 0,C 180,E1 -6426.353,E2 -6426.353} C_VEL
LIN {X 0,Y 488.703,Z 354.238,A -85,B 0,C 180,E1 -6429.255,E2 -6429.255} C_VEL
LIN {X 0,Y 488.702,Z 354.238,A -85,B 0,C 180,E1 -6431.599,E2 -6431.599} C_VEL
LIN {X 0,Y 488.743,Z 354.421,A -85,B 0,C 180,E1 -6435.005,E2 -6435.005} C_VEL
LIN {X 0,Y 491.541,Z 367.235,A -85,B 0,C 180,E1 -6437.302,E2 -6437.302} C_VEL
LIN {X 0,Y 491.543,Z 371.456,A -85,B 0,C 180,E1 -6437.998,E2 -6437.998} C_VEL
LIN {X 0,Y 495.547,Z 389.362,A -85,B 0,C 180,E1 -6438.495,E2 -6438.495} C_VEL
LIN {X 0,Y 493.8,Z 537.21,A -85,B 0,C 180,E1 -6440.817,E2 -6440.817} C_VEL
LIN {X 0,Y 493.407,Z 552.81,A -85,B 0,C 180,E1 -6441.231,E2 -6441.231} C_VEL
LIN {X 0,Y 492.978,Z 566.357,A -85,B 0,C 180,E1 -6441.738,E2 -6441.738} C_VEL
LIN {X 0,Y 492.374,Z 581.095,A -85,B 0,C 180,E1 -6442.46,E2 -6442.46} C_VEL
LIN {X 0,Y 491.732,Z 595.595,A -85,B 0,C 180,E1 -6443.365,E2 -6443.365} C_VEL
LIN {X 0,Y 491.025,Z 608.391,A -85,B 0,C 180,E1 -6444.347,E2 -6444.347} C_VEL
LIN {X 0,Y 490.371,Z 621.006,A -85,B 0,C 180,E1 -6445.52,E2 -6445.52} C_VEL
LIN {X 0,Y 489.807,Z 631.974,A -85,B 0,C 180,E1 -6446.744,E2 -6446.744} C_VEL
LIN {X 0,Y 489.261,Z 642.56,A -85,B 0,C 180,E1 -6448.152,E2 -6448.152} C_VEL
LIN {X 0,Y 488.836,Z 651.686,A -85,B 0,C 180,E1 -6449.613,E2 -6449.613} C_VEL
LIN {X 0,Y 488.496,Z 659.302,A -85,B 0,C 180,E1 -6451.081,E2 -6451.081} C_VEL
LIN {X 0,Y 488.245,Z 665.694,A -85,B 0,C 180,E1 -6452.572,E2 -6452.572} C_VEL
LIN {X 0,Y 488.1,Z 670.546,A -85,B 0,C 180,E1 -6453.949,E2 -6453.949} C_VEL
LIN {X 0,Y 487.94,Z 675.458,A -85,B 0,C 180,E1 -6455.764,E2 -6455.764} C_VEL
LIN {X 0,Y 487.858,Z 678.305,A -85,B 0,C 180,E1 -6457.218,E2 -6457.218} C_VEL
LIN {X 0,Y 487.799,Z 680.417,A -85,B 0,C 180,E1 -6458.888,E2 -6458.888} C_VEL
LIN {X 0,Y 487.777,Z 681.372,A -85,B 0,C 180,E1 -6460.647,E2 -6460.647} C_VEL
LIN {X 0,Y 487.811,Z 681.038,A -85,B 0,C 180,E1 -6462.389,E2 -6462.389} C_VEL
LIN {X 0,Y 487.79,Z 679.455,A -85,B 0,C 180,E1 -6464.112,E2 -6464.112} C_VEL
LIN {X 0,Y 487.877,Z 676.612,A -85,B 0,C 180,E1 -6465.824,E2 -6465.824} C_VEL
LIN {X 0,Y 488.031,Z 672.471,A -85,B 0,C 180,E1 -6467.525,E2 -6467.525} C_VEL
LIN {X 0,Y 488.195,Z 666.971,A -85,B 0,C 180,E1 -6469.213,E2 -6469.213} C_VEL
LIN {X 0,Y 488.472,Z 659.968,A -85,B 0,C 180,E1 -6470.894,E2 -6470.894} C_VEL
LIN {X 0,Y 488.819,Z 652.476,A -85,B 0,C 180,E1 -6472.357,E2 -6472.357} C_VEL
LIN {X 0,Y 489.234,Z 643.475,A -85,B 0,C 180,E1 -6473.815,E2 -6473.815} C_VEL
LIN {X 0,Y 489.767,Z 632.684,A -85,B 0,C 180,E1 -6475.267,E2 -6475.267} C_VEL
LIN {X 0,Y 490.313,Z 621.614,A -85,B 0,C 180,E1 -6476.507,E2 -6476.507} C_VEL
LIN {X 0,Y 490.992,Z 609.479,A -85,B 0,C 180,E1 -6477.641,E2 -6477.641} C_VEL
LIN {X 0,Y 491.676,Z 596.197,A -85,B 0,C 180,E1 -6478.669,E2 -6478.669} C_VEL
LIN {X 0,Y 492.317,Z 581.792,A -85,B 0,C 180,E1 -6479.571,E2 -6479.571} C_VEL
LIN {X 0,Y 492.898,Z 566.804,A -85,B 0,C 180,E1 -6480.306,E2 -6480.306} C_VEL
LIN {X 0,Y 493.38,Z 551.542,A -85,B 0,C 180,E1 -6480.867,E2 -6480.867} C_VEL
LIN {X 0,Y 493.758,Z 536.589,A -85,B 0,C 180,E1 -6481.249,E2 -6481.249} C_VEL
LIN {X 0,Y 495.585,Z 389.201,A -85,B 0,C 180,E1 -6483.618,E2 -6483.618} C_VEL
LIN {X 0,Y 491.794,Z 372.474,A -85,B 0,C 180,E1 -6484.123,E2 -6484.123} C_VEL
LIN {X 0,Y 491.807,Z 367.763,A -85,B 0,C 180,E1 -6484.918,E2 -6484.918} C_VEL
LIN {X 0,Y 489.361,Z 356.508,A -85,B 0,C 180,E1 -6487.02,E2 -6487.02} C_VEL
LIN {X 0,Y 488.821,Z 354.224,A -85,B 0,C 180,E1 -6487.486,E2 -6487.486} C_VEL
LIN {X 0,Y 488.738,Z 354.234,A -85,B 0,C 180,E1 -6490.774,E2 -6490.774} C_VEL
LIN {X 0,Y 488.732,Z 354.231,A -85,B 0,C 180,E1 -6493.302,E2 -6493.302} C_VEL
LIN {X 0,Y 488.764,Z 354.229,A -85,B 0,C 180,E1 -6495.855,E2 -6495.855} C_VEL
LIN {X 0,Y 488.743,Z 354.228,A -85,B 0,C 180,E1 -6499.313,E2 -6499.313} C_VEL
LIN {X 0,Y 488.702,Z 354.235,A -85,B 0,C 180,E1 -6501.956,E2 -6501.956} C_VEL
LIN {X 0,Y 488.702,Z 354.233,A -85,B 0,C 180,E1 -6505.04,E2 -6505.04} C_VEL
LIN {X 0,Y 488.695,Z 354.239,A -85,B 0,C 180,E1 -6508.332,E2 -6508.332} C_VEL
LIN {X 0,Y 488.688,Z 354.233,A -85,B 0,C 180,E1 -6511.18,E2 -6511.18} C_VEL
LIN {X 0,Y 488.719,Z 354.236,A -85,B 0,C 180,E1 -6514.114,E2 -6514.114} C_VEL
LIN {X 0,Y 488.65,Z 354.239,A -85,B 0,C 180,E1 -6517.161,E2 -6517.161} C_VEL
LIN {X 0,Y 488.676,Z 354.235,A -85,B 0,C 180,E1 -6519.256,E2 -6519.256} C_VEL
LIN {X 0,Y 488.65,Z 354.241,A -85,B 0,C 180,E1 -6522.53,E2 -6522.53} C_VEL
LIN {X 0,Y 488.698,Z 354.231,A -85,B 0,C 180,E1 -6525.196,E2 -6525.196} C_VEL
LIN {X 0,Y 488.644,Z 354.24,A -85,B 0,C 180,E1 -6528.577,E2 -6528.577} C_VEL
LIN {X 0,Y 488.651,Z 354.244,A -85,B 0,C 180,E1 -6531.796,E2 -6531.796} C_VEL
LIN {X 0,Y 488.704,Z 354.236,A -85,B 0,C 180,E1 -6535.056,E2 -6535.056} C_VEL
LIN {X 0,Y 488.691,Z 354.243,A -85,B 0,C 180,E1 -6538.048,E2 -6538.048} C_VEL
LIN {X 0,Y 488.715,Z 354.349,A -85,B 0,C 180,E1 -6540.492,E2 -6540.492} C_VEL
LIN {X 0,Y 492.059,Z 368.161,A -85,B 0,C 180,E1 -6542.802,E2 -6542.802} C_VEL
LIN {X 0,Y 492.682,Z 372.821,A -85,B 0,C 180,E1 -6543.526,E2 -6543.526} C_VEL
LIN {X 0,Y 491.549,Z 396.176,A -85,B 0,C 180,E1 -6546.847,E2 -6546.847} C_VEL
LIN {X 0,Y 491.583,Z 397.005,A -85,B 0,C 180,E1 -6546.92,E2 -6546.92} C_VEL
LIN {X 0,Y 495.455,Z 417.237,A -85,B 0,C 180,E1 -6547.46,E2 -6547.46} C_VEL
LIN {X 0,Y 493.86,Z 542.966,A -85,B 0,C 180,E1 -6549.458,E2 -6549.458} C_VEL
LIN {X 0,Y 493.556,Z 565.978,A -85,B 0,C 180,E1 -6549.853,E2 -6549.853} C_VEL
LIN {X 0,Y 493.107,Z 581.294,A -85,B 0,C 180,E1 -6550.276,E2 -6550.276} C_VEL
LIN {X 0,Y 492.606,Z 595.91,A -85,B 0,C 180,E1 -6550.843,E2 -6550.843} C_VEL
LIN {X 0,Y 491.982,Z 610.38,A -85,B 0,C 180,E1 -6551.574,E2 -6551.574} C_VEL
LIN {X 0,Y 491.391,Z 623.638,A -85,B 0,C 180,E1 -6552.413,E2 -6552.413} C_VEL
LIN {X 0,Y 490.762,Z 635.961,A -85,B 0,C 180,E1 -6553.356,E2 -6553.356} C_VEL
LIN {X 0,Y 490.115,Z 648.478,A -85,B 0,C 180,E1 -6554.509,E2 -6554.509} C_VEL
LIN {X 0,Y 489.528,Z 660.719,A -85,B 0,C 180,E1 -6555.872,E2 -6555.872} C_VEL
LIN {X 0,Y 489.053,Z 670.215,A -85,B 0,C 180,E1 -6557.129,E2 -6557.129} C_VEL
LIN {X 0,Y 488.641,Z 679.498,A -85,B 0,C 180,E1 -6558.593,E2 -6558.593} C_VEL
LIN {X 0,Y 488.318,Z 687.189,A -85,B 0,C 180,E1 -6560.054,E2 -6560.054} C_VEL
LIN {X 0,Y 488.133,Z 694.365,A -85,B 0,C 180,E1 -6561.721,E2 -6561.721} C_VEL
LIN {X 0,Y 488,Z 700.575,A -85,B 0,C 180,E1 -6563.571,E2 -6563.571} C_VEL
LIN {X 0,Y 487.928,Z 704.254,A -85,B 0,C 180,E1 -6565.041,E2 -6565.041} C_VEL
LIN {X 0,Y 487.946,Z 707.239,A -85,B 0,C 180,E1 -6566.696,E2 -6566.696} C_VEL
LIN {X 0,Y 487.888,Z 709.025,A -85,B 0,C 180,E1 -6568.348,E2 -6568.348} C_VEL
LIN {X 0,Y 487.816,Z 709.641,A -85,B 0,C 180,E1 -6569.999,E2 -6569.999} C_VEL
LIN {X 0,Y 487.888,Z 709.047,A -85,B 0,C 180,E1 -6571.65,E2 -6571.65} C_VEL
LIN {X 0,Y 487.948,Z 707.288,A -85,B 0,C 180,E1 -6573.302,E2 -6573.302} C_VEL
LIN {X 0,Y 487.928,Z 704.336,A -85,B 0,C 180,E1 -6574.957,E2 -6574.957} C_VEL
LIN {X 0,Y 488.068,Z 700.122,A -85,B 0,C 180,E1 -6576.614,E2 -6576.614} C_VEL
LIN {X 0,Y 488.139,Z 694.527,A -85,B 0,C 180,E1 -6578.277,E2 -6578.277} C_VEL
LIN {X 0,Y 488.319,Z 687.403,A -85,B 0,C 180,E1 -6579.944,E2 -6579.944} C_VEL
LIN {X 0,Y 488.66,Z 679.778,A -85,B 0,C 180,E1 -6581.404,E2 -6581.404} C_VEL
LIN {X 0,Y 489.058,Z 670.585,A -85,B 0,C 180,E1 -6582.869,E2 -6582.869} C_VEL
LIN {X 0,Y 489.631,Z 659.472,A -85,B 0,C 180,E1 -6584.334,E2 -6584.334} C_VEL
LIN {X 0,Y 490.206,Z 648.042,A -85,B 0,C 180,E1 -6585.592,E2 -6585.592} C_VEL
LIN {X 0,Y 490.884,Z 635.475,A -85,B 0,C 180,E1 -6586.745,E2 -6586.745} C_VEL
LIN {X 0,Y 491.517,Z 623.127,A -85,B 0,C 180,E1 -6587.687,E2 -6587.687} C_VEL
LIN {X 0,Y 492.193,Z 609.768,A -85,B 0,C 180,E1 -6588.523,E2 -6588.523} C_VEL
LIN {X 0,Y 492.693,Z 597.401,A -85,B 0,C 180,E1 -6589.151,E2 -6589.151} C_VEL
LIN {X 0,Y 493.234,Z 582.097,A -85,B 0,C 180,E1 -6589.757,E2 -6589.757} C_VEL
LIN {X 0,Y 493.645,Z 567.514,A -85,B 0,C 180,E1 -6590.168,E2 -6590.168} C_VEL
LIN {X 0,Y 493.971,Z 546.625,A -85,B 0,C 180,E1 -6590.535,E2 -6590.535} C_VEL
LIN {X 0,Y 495.371,Z 416.83,A -85,B 0,C 180,E1 -6592.558,E2 -6592.558} C_VEL
LIN {X 0,Y 491.611,Z 397.407,A -85,B 0,C 180,E1 -6593.073,E2 -6593.073} C_VEL
LIN {X 0,Y 492.733,Z 374.923,A -85,B 0,C 180,E1 -6596.24,E2 -6596.24} C_VEL
LIN {X 0,Y 492.779,Z 371.788,A -85,B 0,C 180,E1 -6596.694,E2 -6596.694} C_VEL
LIN {X 0,Y 489.392,Z 357.016,A -85,B 0,C 180,E1 -6599.068,E2 -6599.068} C_VEL
LIN {X 0,Y 488.718,Z 354.235,A -85,B 0,C 180,E1 -6599.565,E2 -6599.565} C_VEL
LIN {X 0,Y 488.727,Z 354.23,A -85,B 0,C 180,E1 -6603.122,E2 -6603.122} C_VEL
LIN {X 0,Y 488.656,Z 354.243,A -85,B 0,C 180,E1 -6606.132,E2 -6606.132} C_VEL
LIN {X 0,Y 488.677,Z 354.235,A -85,B 0,C 180,E1 -6609.254,E2 -6609.254} C_VEL
LIN {X 0,Y 488.656,Z 354.24,A -85,B 0,C 180,E1 -6612.527,E2 -6612.527} C_VEL
LIN {X 0,Y 488.689,Z 354.232,A -85,B 0,C 180,E1 -6615.196,E2 -6615.196} C_VEL
LIN {X 0,Y 488.649,Z 354.24,A -85,B 0,C 180,E1 -6618.579,E2 -6618.579} C_VEL
LIN {X 0,Y 488.675,Z 354.234,A -85,B 0,C 180,E1 -6620.949,E2 -6620.949} C_VEL
LIN {X 0,Y 488.639,Z 354.243,A -85,B 0,C 180,E1 -6623.865,E2 -6623.865} C_VEL
LIN {X 0,Y 488.723,Z 354.228,A -85,B 0,C 180,E1 -6626.876,E2 -6626.876} C_VEL
LIN {X 0,Y 488.704,Z 354.234,A -85,B 0,C 180,E1 -6629.78,E2 -6629.78} C_VEL
LIN {X 0,Y 488.682,Z 354.233,A -85,B 0,C 180,E1 -6633.078,E2 -6633.078} C_VEL
LIN {X 0,Y 488.654,Z 354.243,A -85,B 0,C 180,E1 -6636.253,E2 -6636.253} C_VEL
LIN {X 0,Y 488.731,Z 354.226,A -85,B 0,C 180,E1 -6639.175,E2 -6639.175} C_VEL
LIN {X 0,Y 488.731,Z 354.229,A -85,B 0,C 180,E1 -6641.632,E2 -6641.632} C_VEL
LIN {X 0,Y 488.732,Z 354.226,A -85,B 0,C 180,E1 -6644.999,E2 -6644.999} C_VEL
LIN {X 0,Y 488.789,Z 354.223,A -85,B 0,C 180,E1 -6648.387,E2 -6648.387} C_VEL
LIN {X 0,Y 488.746,Z 354.229,A -85,B 0,C 180,E1 -6651.733,E2 -6651.733} C_VEL
LIN {X 0,Y 488.802,Z 354.223,A -85,B 0,C 180,E1 -6654.224,E2 -6654.224} C_VEL
LIN {X 0,Y 488.926,Z 354.205,A -85,B 0,C 180,E1 -6657.529,E2 -6657.529} C_VEL
LIN {X 0,Y 488.925,Z 354.211,A -85,B 0,C 180,E1 -6660,E2 -6660} C_VEL
LIN {X 0,Y 488.925,Z 354.205,A -85,B 0,C 180,E1 -6662.472,E2 -6662.472} C_VEL
LIN {X 0,Y 488.797,Z 354.224,A -85,B 0,C 180,E1 -6665.777,E2 -6665.777} C_VEL
LIN {X 0,Y 488.744,Z 354.229,A -85,B 0,C 180,E1 -6668.268,E2 -6668.268} C_VEL
LIN {X 0,Y 488.768,Z 354.226,A -85,B 0,C 180,E1 -6671.614,E2 -6671.614} C_VEL
LIN {X 0,Y 488.733,Z 354.226,A -85,B 0,C 180,E1 -6675.002,E2 -6675.002} C_VEL
LIN {X 0,Y 488.729,Z 354.229,A -85,B 0,C 180,E1 -6678.443,E2 -6678.443} C_VEL
LIN {X 0,Y 488.692,Z 354.231,A -85,B 0,C 180,E1 -6681.072,E2 -6681.072} C_VEL
LIN {X 0,Y 488.655,Z 354.242,A -85,B 0,C 180,E1 -6683.748,E2 -6683.748} C_VEL
LIN {X 0,Y 488.683,Z 354.232,A -85,B 0,C 180,E1 -6686.922,E2 -6686.922} C_VEL
LIN {X 0,Y 488.705,Z 354.234,A -85,B 0,C 180,E1 -6690.221,E2 -6690.221} C_VEL
LIN {X 0,Y 488.719,Z 354.231,A -85,B 0,C 180,E1 -6693.485,E2 -6693.485} C_VEL
LIN {X 0,Y 488.644,Z 354.24,A -85,B 0,C 180,E1 -6696.351,E2 -6696.351} C_VEL
LIN {X 0,Y 488.677,Z 354.235,A -85,B 0,C 180,E1 -6699.257,E2 -6699.257} C_VEL
LIN {X 0,Y 488.657,Z 354.241,A -85,B 0,C 180,E1 -6701.596,E2 -6701.596} C_VEL
LIN {X 0,Y 488.692,Z 354.231,A -85,B 0,C 180,E1 -6704.804,E2 -6704.804} C_VEL
LIN {X 0,Y 488.658,Z 354.239,A -85,B 0,C 180,E1 -6707.473,E2 -6707.473} C_VEL
LIN {X 0,Y 488.68,Z 354.233,A -85,B 0,C 180,E1 -6710.746,E2 -6710.746} C_VEL
LIN {X 0,Y 488.658,Z 354.243,A -85,B 0,C 180,E1 -6713.868,E2 -6713.868} C_VEL
LIN {X 0,Y 488.73,Z 354.227,A -85,B 0,C 180,E1 -6716.878,E2 -6716.878} C_VEL
LIN {X 0,Y 488.714,Z 354.238,A -85,B 0,C 180,E1 -6719.782,E2 -6719.782} C_VEL
LIN {X 0,Y 488.693,Z 354.232,A -85,B 0,C 180,E1 -6723.08,E2 -6723.08} C_VEL
LIN {X 0,Y 488.654,Z 354.237,A -85,B 0,C 180,E1 -6724.311,E2 -6724.311} C_VEL
LIN {X 0,Y 488.011,Z 354.319,A -85,B 0,C 180,E1 -6724.999,E2 -6724.999} C_VEL
LIN {X 0,Y 485.179,Z 354.679,A -85,B 0,C 180,E1 -6726.117,E2 -6726.117} C_VEL
LIN {X 0,Y 482.767,Z 354.981,A -85,B 0,C 180,E1 -6727.018,E2 -6727.018} C_VEL
LIN {X 0,Y 481.723,Z 355.108,A -85,B 0,C 180,E1 -6727.714,E2 -6727.714} C_VEL
LIN {X 0,Y 481.635,Z 355.115,A -85,B 0,C 180,E1 -6727.949,E2 -6727.949} C_VEL
LIN {X 0,Y 481.699,Z 355.103,A -85,B 0,C 180,E1 -6730.394,E2 -6730.394} C_VEL
LIN {X 0,Y 481.664,Z 355.108,A -85,B 0,C 180,E1 -6733.034,E2 -6733.034} C_VEL
LIN {X 0,Y 481.682,Z 355.112,A -85,B 0,C 180,E1 -6735.64,E2 -6735.64} C_VEL
LIN {X 0,Y 481.752,Z 355.098,A -85,B 0,C 180,E1 -6738.217,E2 -6738.217} C_VEL
LIN {X 0,Y 481.722,Z 355.107,A -85,B 0,C 180,E1 -6741.612,E2 -6741.612} C_VEL
LIN {X 0,Y 481.777,Z 355.095,A -85,B 0,C 180,E1 -6744.14,E2 -6744.14} C_VEL
LIN {X 0,Y 481.911,Z 355.082,A -85,B 0,C 180,E1 -6747.494,E2 -6747.494} C_VEL
LIN {X 0,Y 481.914,Z 355.08,A -85,B 0,C 180,E1 -6750.001,E2 -6750.001} C_VEL
LIN {X 0,Y 481.912,Z 355.076,A -85,B 0,C 180,E1 -6752.509,E2 -6752.509} C_VEL
LIN {X 0,Y 481.781,Z 355.098,A -85,B 0,C 180,E1 -6755.862,E2 -6755.862} C_VEL
LIN {X 0,Y 481.74,Z 355.098,A -85,B 0,C 180,E1 -6758.39,E2 -6758.39} C_VEL
LIN {X 0,Y 481.756,Z 355.101,A -85,B 0,C 180,E1 -6761.786,E2 -6761.786} C_VEL
LIN {X 0,Y 481.736,Z 355.101,A -85,B 0,C 180,E1 -6765.225,E2 -6765.225} C_VEL
LIN {X 0,Y 481.712,Z 355.101,A -85,B 0,C 180,E1 -6768.723,E2 -6768.723} C_VEL
LIN {X 0,Y 481.652,Z 355.114,A -85,B 0,C 180,E1 -6771.396,E2 -6771.396} C_VEL
LIN {X 0,Y 481.654,Z 355.11,A -85,B 0,C 180,E1 -6774.115,E2 -6774.115} C_VEL
LIN {X 0,Y 481.659,Z 355.11,A -85,B 0,C 180,E1 -6777.118,E2 -6777.118} C_VEL
LIN {X 0,Y 481.673,Z 355.111,A -85,B 0,C 180,E1 -6779.743,E2 -6779.743} C_VEL
LIN {X 0,Y 481.678,Z 355.105,A -85,B 0,C 180,E1 -6782.675,E2 -6782.675} C_VEL
LIN {X 0,Y 481.637,Z 355.118,A -85,B 0,C 180,E1 -6785.711,E2 -6785.711} C_VEL
LIN {X 0,Y 481.674,Z 355.11,A -85,B 0,C 180,E1 -6788.86,E2 -6788.86} C_VEL
LIN {X 0,Y 481.652,Z 355.116,A -85,B 0,C 180,E1 -6791.912,E2 -6791.912} C_VEL
LIN {X 0,Y 481.691,Z 355.224,A -85,B 0,C 180,E1 -6794.712,E2 -6794.712} C_VEL
LIN {X 0,Y 484.711,Z 369.158,A -85,B 0,C 180,E1 -6797.249,E2 -6797.249} C_VEL
LIN {X 0,Y 484.742,Z 371.612,A -85,B 0,C 180,E1 -6797.66,E2 -6797.66} C_VEL
LIN {X 0,Y 488.924,Z 390.189,A -85,B 0,C 180,E1 -6798.19,E2 -6798.19} C_VEL
LIN {X 0,Y 487.141,Z 536.616,A -85,B 0,C 180,E1 -6800.532,E2 -6800.532} C_VEL
LIN {X 0,Y 486.706,Z 552.425,A -85,B 0,C 180,E1 -6800.949,E2 -6800.949} C_VEL
LIN {X 0,Y 486.215,Z 566.492,A -85,B 0,C 180,E1 -6801.48,E2 -6801.48} C_VEL
LIN {X 0,Y 485.564,Z 581.667,A -85,B 0,C 180,E1 -6802.234,E2 -6802.234} C_VEL
LIN {X 0,Y 484.928,Z 595.174,A -85,B 0,C 180,E1 -6803.088,E2 -6803.088} C_VEL
LIN {X 0,Y 484.14,Z 609.093,A -85,B 0,C 180,E1 -6804.169,E2 -6804.169} C_VEL
LIN {X 0,Y 483.463,Z 621.413,A -85,B 0,C 180,E1 -6805.336,E2 -6805.336} C_VEL
LIN {X 0,Y 482.806,Z 633.076,A -85,B 0,C 180,E1 -6806.666,E2 -6806.666} C_VEL
LIN {X 0,Y 482.229,Z 643.783,A -85,B 0,C 180,E1 -6808.138,E2 -6808.138} C_VEL
LIN {X 0,Y 481.783,Z 652.662,A -85,B 0,C 180,E1 -6809.601,E2 -6809.601} C_VEL
LIN {X 0,Y 481.412,Z 660.672,A -85,B 0,C 180,E1 -6811.199,E2 -6811.199} C_VEL
LIN {X 0,Y 481.131,Z 667.91,A -85,B 0,C 180,E1 -6813.006,E2 -6813.006} C_VEL
LIN {X 0,Y 480.977,Z 672.544,A -85,B 0,C 180,E1 -6814.465,E2 -6814.465} C_VEL
LIN {X 0,Y 480.839,Z 675.968,A -85,B 0,C 180,E1 -6815.842,E2 -6815.842} C_VEL
LIN {X 0,Y 480.749,Z 679.23,A -85,B 0,C 180,E1 -6817.66,E2 -6817.66} C_VEL
LIN {X 0,Y 480.757,Z 681.088,A -85,B 0,C 180,E1 -6819.461,E2 -6819.461} C_VEL
LIN {X 0,Y 480.708,Z 681.621,A -85,B 0,C 180,E1 -6821.237,E2 -6821.237} C_VEL
LIN {X 0,Y 480.693,Z 680.879,A -85,B 0,C 180,E1 -6822.997,E2 -6822.997} C_VEL
LIN {X 0,Y 480.763,Z 678.848,A -85,B 0,C 180,E1 -6824.759,E2 -6824.759} C_VEL
LIN {X 0,Y 480.831,Z 675.572,A -85,B 0,C 180,E1 -6826.475,E2 -6826.475} C_VEL
LIN {X 0,Y 481.051,Z 670.948,A -85,B 0,C 180,E1 -6828.197,E2 -6828.197} C_VEL
LIN {X 0,Y 481.21,Z 664.947,A -85,B 0,C 180,E1 -6829.906,E2 -6829.906} C_VEL
LIN {X 0,Y 481.547,Z 657.392,A -85,B 0,C 180,E1 -6831.608,E2 -6831.608} C_VEL
LIN {X 0,Y 481.945,Z 649.3,A -85,B 0,C 180,E1 -6833.091,E2 -6833.091} C_VEL
LIN {X 0,Y 482.439,Z 639.635,A -85,B 0,C 180,E1 -6834.566,E2 -6834.566} C_VEL
LIN {X 0,Y 482.968,Z 629.776,A -85,B 0,C 180,E1 -6835.827,E2 -6835.827} C_VEL
LIN {X 0,Y 483.65,Z 618.081,A -85,B 0,C 180,E1 -6837.084,E2 -6837.084} C_VEL
LIN {X 0,Y 484.35,Z 605.228,A -85,B 0,C 180,E1 -6838.233,E2 -6838.233} C_VEL
LIN {X 0,Y 485.032,Z 592.499,A -85,B 0,C 180,E1 -6839.17,E2 -6839.17} C_VEL
LIN {X 0,Y 485.67,Z 578.639,A -85,B 0,C 180,E1 -6840,E2 -6840} C_VEL
LIN {X 0,Y 486.222,Z 564.392,A -85,B 0,C 180,E1 -6840.673,E2 -6840.673} C_VEL
LIN {X 0,Y 486.716,Z 549.011,A -85,B 0,C 180,E1 -6841.215,E2 -6841.215} C_VEL
LIN {X 0,Y 487.092,Z 533.861,A -85,B 0,C 180,E1 -6841.576,E2 -6841.576} C_VEL
LIN {X 0,Y 489.056,Z 391.266,A -85,B 0,C 180,E1 -6843.914,E2 -6843.914} C_VEL
LIN {X 0,Y 487.841,Z 384.64,A -85,B 0,C 180,E1 -6844.098,E2 -6844.098} C_VEL
LIN {X 0,Y 485.055,Z 372.814,A -85,B 0,C 180,E1 -6844.477,E2 -6844.477} C_VEL
LIN {X 0,Y 485.049,Z 369.858,A -85,B 0,C 180,E1 -6844.987,E2 -6844.987} C_VEL
LIN {X 0,Y 482.88,Z 359.569,A -85,B 0,C 180,E1 -6846.936,E2 -6846.936} C_VEL
LIN {X 0,Y 481.762,Z 355.103,A -85,B 0,C 180,E1 -6847.829,E2 -6847.829} C_VEL
LIN {X 0,Y 481.707,Z 355.108,A -85,B 0,C 180,E1 -6850.933,E2 -6850.933} C_VEL
LIN {X 0,Y 481.696,Z 355.108,A -85,B 0,C 180,E1 -6853.5,E2 -6853.5} C_VEL
LIN {X 0,Y 481.697,Z 355.111,A -85,B 0,C 180,E1 -6856.094,E2 -6856.094} C_VEL
LIN {X 0,Y 481.712,Z 355.108,A -85,B 0,C 180,E1 -6858.722,E2 -6858.722} C_VEL
LIN {X 0,Y 481.65,Z 355.111,A -85,B 0,C 180,E1 -6861.394,E2 -6861.394} C_VEL
LIN {X 0,Y 481.652,Z 355.115,A -85,B 0,C 180,E1 -6864.114,E2 -6864.114} C_VEL
LIN {X 0,Y 481.654,Z 355.111,A -85,B 0,C 180,E1 -6867.116,E2 -6867.116} C_VEL
LIN {X 0,Y 481.668,Z 355.111,A -85,B 0,C 180,E1 -6869.742,E2 -6869.742} C_VEL
LIN {X 0,Y 481.654,Z 355.113,A -85,B 0,C 180,E1 -6872.675,E2 -6872.675} C_VEL
LIN {X 0,Y 481.651,Z 355.111,A -85,B 0,C 180,E1 -6875.201,E2 -6875.201} C_VEL
LIN {X 0,Y 481.631,Z 355.118,A -85,B 0,C 180,E1 -6878.002,E2 -6878.002} C_VEL
LIN {X 0,Y 481.606,Z 355.116,A -85,B 0,C 180,E1 -6881.047,E2 -6881.047} C_VEL
LIN {X 0,Y 481.652,Z 355.112,A -85,B 0,C 180,E1 -6884.458,E2 -6884.458} C_VEL
LIN {X 0,Y 481.614,Z 355.115,A -85,B 0,C 180,E1 -6886.855,E2 -6886.855} C_VEL
LIN {X 0,Y 481.63,Z 355.118,A -85,B 0,C 180,E1 -6890.054,E2 -6890.054} C_VEL
LIN {X 0,Y 481.605,Z 355.119,A -85,B 0,C 180,E1 -6893.25,E2 -6893.25} C_VEL
LIN {X 0,Y 481.673,Z 355.115,A -85,B 0,C 180,E1 -6896.326,E2 -6896.326} C_VEL
LIN {X 0,Y 481.661,Z 355.119,A -85,B 0,C 180,E1 -6899.774,E2 -6899.774} C_VEL
LIN {X 0,Y 481.682,Z 355.233,A -85,B 0,C 180,E1 -6900.138,E2 -6900.138} C_VEL
LIN {X 0,Y 485.178,Z 369.705,A -85,B 0,C 180,E1 -6902.618,E2 -6902.618} C_VEL
LIN {X 0,Y 485.882,Z 374.312,A -85,B 0,C 180,E1 -6903.358,E2 -6903.358} C_VEL
LIN {X 0,Y 484.767,Z 396.266,A -85,B 0,C 180,E1 -6906.535,E2 -6906.535} C_VEL
LIN {X 0,Y 488.928,Z 418.583,A -85,B 0,C 180,E1 -6907.162,E2 -6907.162} C_VEL
LIN {X 0,Y 486.885,Z 563.822,A -85,B 0,C 180,E1 -6909.537,E2 -6909.537} C_VEL
LIN {X 0,Y 486.381,Z 579.919,A -85,B 0,C 180,E1 -6909.971,E2 -6909.971} C_VEL
LIN {X 0,Y 485.835,Z 595.223,A -85,B 0,C 180,E1 -6910.565,E2 -6910.565} C_VEL
LIN {X 0,Y 485.189,Z 609.77,A -85,B 0,C 180,E1 -6911.307,E2 -6911.307} C_VEL
LIN {X 0,Y 484.562,Z 623.085,A -85,B 0,C 180,E1 -6912.157,E2 -6912.157} C_VEL
LIN {X 0,Y 483.881,Z 635.443,A -85,B 0,C 180,E1 -6913.112,E2 -6913.112} C_VEL
LIN {X 0,Y 483.208,Z 648.022,A -85,B 0,C 180,E1 -6914.282,E2 -6914.282} C_VEL
LIN {X 0,Y 482.57,Z 660.319,A -85,B 0,C 180,E1 -6915.664,E2 -6915.664} C_VEL
LIN {X 0,Y 482.052,Z 669.84,A -85,B 0,C 180,E1 -6916.938,E2 -6916.938} C_VEL
LIN {X 0,Y 481.61,Z 679.159,A -85,B 0,C 180,E1 -6918.424,E2 -6918.424} C_VEL
LIN {X 0,Y 481.272,Z 686.885,A -85,B 0,C 180,E1 -6919.906,E2 -6919.906} C_VEL
LIN {X 0,Y 481.059,Z 694.089,A -85,B 0,C 180,E1 -6921.598,E2 -6921.598} C_VEL
LIN {X 0,Y 480.908,Z 699.747,A -85,B 0,C 180,E1 -6923.285,E2 -6923.285} C_VEL
LIN {X 0,Y 480.853,Z 704.023,A -85,B 0,C 180,E1 -6924.968,E2 -6924.968} C_VEL
LIN {X 0,Y 480.851,Z 707.022,A -85,B 0,C 180,E1 -6926.647,E2 -6926.647} C_VEL
LIN {X 0,Y 480.818,Z 708.815,A -85,B 0,C 180,E1 -6928.324,E2 -6928.324} C_VEL
LIN {X 0,Y 480.74,Z 709.437,A -85,B 0,C 180,E1 -6929.999,E2 -6929.999} C_VEL
LIN {X 0,Y 480.818,Z 708.843,A -85,B 0,C 180,E1 -6931.674,E2 -6931.674} C_VEL
LIN {X 0,Y 480.871,Z 707.08,A -85,B 0,C 180,E1 -6933.35,E2 -6933.35} C_VEL
LIN {X 0,Y 480.854,Z 704.118,A -85,B 0,C 180,E1 -6935.03,E2 -6935.03} C_VEL
LIN {X 0,Y 480.969,Z 699.893,A -85,B 0,C 180,E1 -6936.712,E2 -6936.712} C_VEL
LIN {X 0,Y 481.066,Z 694.282,A -85,B 0,C 180,E1 -6938.399,E2 -6938.399} C_VEL
LIN {X 0,Y 481.272,Z 687.139,A -85,B 0,C 180,E1 -6940.091,E2 -6940.091} C_VEL
LIN {X 0,Y 481.64,Z 679.492,A -85,B 0,C 180,E1 -6941.573,E2 -6941.573} C_VEL
LIN {X 0,Y 482.063,Z 670.275,A -85,B 0,C 180,E1 -6943.059,E2 -6943.059} C_VEL
LIN {X 0,Y 482.669,Z 659.127,A -85,B 0,C 180,E1 -6944.545,E2 -6944.545} C_VEL
LIN {X 0,Y 483.317,Z 647.663,A -85,B 0,C 180,E1 -6945.82,E2 -6945.82} C_VEL
LIN {X 0,Y 483.983,Z 635.049,A -85,B 0,C 180,E1 -6946.991,E2 -6946.991} C_VEL
LIN {X 0,Y 484.686,Z 622.667,A -85,B 0,C 180,E1 -6947.945,E2 -6947.945} C_VEL
LIN {X 0,Y 485.392,Z 609.254,A -85,B 0,C 180,E1 -6948.792,E2 -6948.792} C_VEL
LIN {X 0,Y 485.936,Z 596.794,A -85,B 0,C 180,E1 -6949.428,E2 -6949.428} C_VEL
LIN {X 0,Y 486.493,Z 581.648,A -85,B 0,C 180,E1 -6950.031,E2 -6950.031} C_VEL
LIN {X 0,Y 486.965,Z 566.512,A -85,B 0,C 180,E1 -6950.457,E2 -6950.457} C_VEL
LIN {X 0,Y 487.324,Z 543.493,A -85,B 0,C 180,E1 -6950.855,E2 -6950.855} C_VEL
LIN {X 0,Y 488.902,Z 418.526,A -85,B 0,C 180,E1 -6952.836,E2 -6952.836} C_VEL
LIN {X 0,Y 484.8,Z 397.212,A -85,B 0,C 180,E1 -6953.416,E2 -6953.416} C_VEL
LIN {X 0,Y 485.956,Z 374.724,A -85,B 0,C 180,E1 -6956.635,E2 -6956.635} C_VEL
LIN {X 0,Y 485.592,Z 371.562,A -85,B 0,C 180,E1 -6957.121,E2 -6957.121} C_VEL
LIN {X 0,Y 482.122,Z 356.915,A -85,B 0,C 180,E1 -6959.527,E2 -6959.527} C_VEL
LIN {X 0,Y 481.669,Z 355.113,A -85,B 0,C 180,E1 -6959.86,E2 -6959.86} C_VEL
LIN {X 0,Y 481.662,Z 355.113,A -85,B 0,C 180,E1 -6962.673,E2 -6962.673} C_VEL
LIN {X 0,Y 481.619,Z 355.117,A -85,B 0,C 180,E1 -6965.709,E2 -6965.709} C_VEL
LIN {X 0,Y 481.622,Z 355.115,A -85,B 0,C 180,E1 -6968.862,E2 -6968.862} C_VEL
LIN {X 0,Y 481.623,Z 355.116,A -85,B 0,C 180,E1 -6971.909,E2 -6971.909} C_VEL
LIN {X 0,Y 481.642,Z 355.114,A -85,B 0,C 180,E1 -6974.457,E2 -6974.457} C_VEL
LIN {X 0,Y 481.611,Z 355.117,A -85,B 0,C 180,E1 -6977.836,E2 -6977.836} C_VEL
LIN {X 0,Y 481.636,Z 355.113,A -85,B 0,C 180,E1 -6980.655,E2 -6980.655} C_VEL
LIN {X 0,Y 481.597,Z 355.116,A -85,B 0,C 180,E1 -6983.378,E2 -6983.378} C_VEL
LIN {X 0,Y 481.68,Z 355.111,A -85,B 0,C 180,E1 -6986.328,E2 -6986.328} C_VEL
LIN {X 0,Y 481.631,Z 355.112,A -85,B 0,C 180,E1 -6989.418,E2 -6989.418} C_VEL
LIN {X 0,Y 481.634,Z 355.119,A -85,B 0,C 180,E1 -6992.164,E2 -6992.164} C_VEL
LIN {X 0,Y 481.658,Z 355.108,A -85,B 0,C 180,E1 -6994.967,E2 -6994.967} C_VEL
LIN {X 0,Y 481.631,Z 355.114,A -85,B 0,C 180,E1 -6997.704,E2 -6997.704} C_VEL
LIN {X 0,Y 481.681,Z 355.109,A -85,B 0,C 180,E1 -7000.392,E2 -7000.392} C_VEL
LIN {X 0,Y 481.602,Z 355.114,A -85,B 0,C 180,E1 -7003.031,E2 -7003.031} C_VEL
LIN {X 0,Y 481.66,Z 355.11,A -85,B 0,C 180,E1 -7005.638,E2 -7005.638} C_VEL
LIN {X 0,Y 481.735,Z 355.104,A -85,B 0,C 180,E1 -7008.215,E2 -7008.215} C_VEL
LIN {X 0,Y 481.705,Z 355.105,A -85,B 0,C 180,E1 -7011.611,E2 -7011.611} C_VEL
LIN {X 0,Y 481.763,Z 355.102,A -85,B 0,C 180,E1 -7014.139,E2 -7014.139} C_VEL
LIN {X 0,Y 481.891,Z 355.081,A -85,B 0,C 180,E1 -7017.493,E2 -7017.493} C_VEL
LIN {X 0,Y 481.894,Z 355.087,A -85,B 0,C 180,E1 -7020,E2 -7020} C_VEL
LIN {X 0,Y 481.891,Z 355.081,A -85,B 0,C 180,E1 -7022.508,E2 -7022.508} C_VEL
LIN {X 0,Y 481.758,Z 355.102,A -85,B 0,C 180,E1 -7025.861,E2 -7025.861} C_VEL
LIN {X 0,Y 481.703,Z 355.105,A -85,B 0,C 180,E1 -7028.39,E2 -7028.39} C_VEL
LIN {X 0,Y 481.72,Z 355.106,A -85,B 0,C 180,E1 -7031.786,E2 -7031.786} C_VEL
LIN {X 0,Y 481.715,Z 355.101,A -85,B 0,C 180,E1 -7035.225,E2 -7035.225} C_VEL
LIN {X 0,Y 481.69,Z 355.104,A -85,B 0,C 180,E1 -7038.723,E2 -7038.723} C_VEL
LIN {X 0,Y 481.63,Z 355.113,A -85,B 0,C 180,E1 -7041.396,E2 -7041.396} C_VEL
LIN {X 0,Y 481.634,Z 355.116,A -85,B 0,C 180,E1 -7044.116,E2 -7044.116} C_VEL
LIN {X 0,Y 481.638,Z 355.11,A -85,B 0,C 180,E1 -7047.118,E2 -7047.118} C_VEL
LIN {X 0,Y 481.653,Z 355.115,A -85,B 0,C 180,E1 -7049.743,E2 -7049.743} C_VEL
LIN {X 0,Y 481.659,Z 355.108,A -85,B 0,C 180,E1 -7052.676,E2 -7052.676} C_VEL
LIN {X 0,Y 481.61,Z 355.12,A -85,B 0,C 180,E1 -7055.712,E2 -7055.712} C_VEL
LIN {X 0,Y 481.621,Z 355.112,A -85,B 0,C 180,E1 -7058.864,E2 -7058.864} C_VEL
LIN {X 0,Y 481.611,Z 355.121,A -85,B 0,C 180,E1 -7061.91,E2 -7061.91} C_VEL
LIN {X 0,Y 481.644,Z 355.11,A -85,B 0,C 180,E1 -7064.46,E2 -7064.46} C_VEL
LIN {X 0,Y 481.617,Z 355.121,A -85,B 0,C 180,E1 -7067.838,E2 -7067.838} C_VEL
LIN {X 0,Y 481.641,Z 355.11,A -85,B 0,C 180,E1 -7070.657,E2 -7070.657} C_VEL
LIN {X 0,Y 481.611,Z 355.116,A -85,B 0,C 180,E1 -7073.379,E2 -7073.379} C_VEL
LIN {X 0,Y 481.665,Z 355.109,A -85,B 0,C 180,E1 -7076.328,E2 -7076.328} C_VEL
LIN {X 0,Y 481.641,Z 355.113,A -85,B 0,C 180,E1 -7079.42,E2 -7079.42} C_VEL
LIN {X 0,Y 481.644,Z 355.113,A -85,B 0,C 180,E1 -7082.166,E2 -7082.166} C_VEL
LIN {X 0,Y 481.669,Z 355.107,A -85,B 0,C 180,E1 -7084.969,E2 -7084.969} C_VEL
LIN {X 0,Y 481.635,Z 355.115,A -85,B 0,C 180,E1 -7087.949,E2 -7087.949} C_VEL
LIN {X 0,Y 480.967,Z 355.196,A -85,B 0,C 180,E1 -7088.647,E2 -7088.647} C_VEL
LIN {X 0,Y 478.144,Z 355.553,A -85,B 0,C 180,E1 -7089.782,E2 -7089.782} C_VEL
LIN {X 0,Y 475.758,Z 355.848,A -85,B 0,C 180,E1 -7090.696,E2 -7090.696} C_VEL
LIN {X 0,Y 474.729,Z 355.975,A -85,B 0,C 180,E1 -7091.402,E2 -7091.402} C_VEL
LIN {X 0,Y 474.642,Z 355.986,A -85,B 0,C 180,E1 -7091.641,E2 -7091.641} C_VEL
LIN {X 0,Y 474.698,Z 355.975,A -85,B 0,C 180,E1 -7094.546,E2 -7094.546} C_VEL
LIN {X 0,Y 474.705,Z 355.978,A -85,B 0,C 180,E1 -7098.039,E2 -7098.039} C_VEL
LIN {X 0,Y 474.698,Z 355.98,A -85,B 0,C 180,E1 -7101.487,E2 -7101.487} C_VEL
LIN {X 0,Y 474.74,Z 355.973,A -85,B 0,C 180,E1 -7104.053,E2 -7104.053} C_VEL
LIN {X 0,Y 474.876,Z 355.958,A -85,B 0,C 180,E1 -7107.457,E2 -7107.457} C_VEL
LIN {X 0,Y 474.883,Z 355.955,A -85,B 0,C 180,E1 -7110.001,E2 -7110.001} C_VEL
LIN {X 0,Y 474.877,Z 355.952,A -85,B 0,C 180,E1 -7112.546,E2 -7112.546} C_VEL
LIN {X 0,Y 474.744,Z 355.973,A -85,B 0,C 180,E1 -7115.949,E2 -7115.949} C_VEL
LIN {X 0,Y 474.712,Z 355.973,A -85,B 0,C 180,E1 -7118.515,E2 -7118.515} C_VEL
LIN {X 0,Y 474.71,Z 355.977,A -85,B 0,C 180,E1 -7121.963,E2 -7121.963} C_VEL
LIN {X 0,Y 474.694,Z 355.982,A -85,B 0,C 180,E1 -7125.457,E2 -7125.457} C_VEL
LIN {X 0,Y 474.666,Z 355.98,A -85,B 0,C 180,E1 -7129.011,E2 -7129.011} C_VEL
LIN {X 0,Y 474.594,Z 355.994,A -85,B 0,C 180,E1 -7131.73,E2 -7131.73} C_VEL
LIN {X 0,Y 474.632,Z 355.983,A -85,B 0,C 180,E1 -7134.495,E2 -7134.495} C_VEL
LIN {X 0,Y 474.606,Z 355.991,A -85,B 0,C 180,E1 -7137.327,E2 -7137.327} C_VEL
LIN {X 0,Y 474.603,Z 355.987,A -85,B 0,C 180,E1 -7140.231,E2 -7140.231} C_VEL
LIN {X 0,Y 474.641,Z 355.986,A -85,B 0,C 180,E1 -7143.221,E2 -7143.221} C_VEL
LIN {X 0,Y 474.59,Z 355.992,A -85,B 0,C 180,E1 -7146.325,E2 -7146.325} C_VEL
LIN {X 0,Y 474.63,Z 355.992,A -85,B 0,C 180,E1 -7149.548,E2 -7149.548} C_VEL
LIN {X 0,Y 474.606,Z 355.992,A -85,B 0,C 180,E1 -7152.234,E2 -7152.234} C_VEL
LIN {X 0,Y 474.665,Z 356.185,A -85,B 0,C 180,E1 -7154.447,E2 -7154.447} C_VEL
LIN {X 0,Y 477.79,Z 370.216,A -85,B 0,C 180,E1 -7157.038,E2 -7157.038} C_VEL
LIN {X 0,Y 477.949,Z 372.1,A -85,B 0,C 180,E1 -7157.327,E2 -7157.327} C_VEL
LIN {X 0,Y 482.38,Z 391.349,A -85,B 0,C 180,E1 -7157.887,E2 -7157.887} C_VEL
LIN {X 0,Y 480.42,Z 537.512,A -85,B 0,C 180,E1 -7160.272,E2 -7160.272} C_VEL
LIN {X 0,Y 479.981,Z 552.471,A -85,B 0,C 180,E1 -7160.674,E2 -7160.674} C_VEL
LIN {X 0,Y 479.427,Z 567.688,A -85,B 0,C 180,E1 -7161.261,E2 -7161.261} C_VEL
LIN {X 0,Y 478.744,Z 582.643,A -85,B 0,C 180,E1 -7162.03,E2 -7162.03} C_VEL
LIN {X 0,Y 478.05,Z 596.523,A -85,B 0,C 180,E1 -7162.932,E2 -7162.932} C_VEL
LIN {X 0,Y 477.286,Z 608.948,A -85,B 0,C 180,E1 -7163.914,E2 -7163.914} C_VEL
LIN {X 0,Y 476.577,Z 621.662,A -85,B 0,C 180,E1 -7165.134,E2 -7165.134} C_VEL
LIN {X 0,Y 475.904,Z 632.462,A -85,B 0,C 180,E1 -7166.372,E2 -7166.372} C_VEL
LIN {X 0,Y 475.282,Z 643.152,A -85,B 0,C 180,E1 -7167.836,E2 -7167.836} C_VEL
LIN {X 0,Y 474.778,Z 652.905,A -85,B 0,C 180,E1 -7169.458,E2 -7169.458} C_VEL
LIN {X 0,Y 474.393,Z 660.266,A -85,B 0,C 180,E1 -7170.936,E2 -7170.936} C_VEL
LIN {X 0,Y 474.082,Z 667.801,A -85,B 0,C 180,E1 -7172.808,E2 -7172.808} C_VEL
LIN {X 0,Y 473.905,Z 673.17,A -85,B 0,C 180,E1 -7174.528,E2 -7174.528} C_VEL
LIN {X 0,Y 473.723,Z 677.446,A -85,B 0,C 180,E1 -7176.386,E2 -7176.386} C_VEL
LIN {X 0,Y 473.623,Z 680.236,A -85,B 0,C 180,E1 -7178.224,E2 -7178.224} C_VEL
LIN {X 0,Y 473.63,Z 681.642,A -85,B 0,C 180,E1 -7180.044,E2 -7180.044} C_VEL
LIN {X 0,Y 473.623,Z 681.72,A -85,B 0,C 180,E1 -7181.843,E2 -7181.843} C_VEL
LIN {X 0,Y 473.608,Z 680.527,A -85,B 0,C 180,E1 -7183.623,E2 -7183.623} C_VEL
LIN {X 0,Y 473.685,Z 678.073,A -85,B 0,C 180,E1 -7185.39,E2 -7185.39} C_VEL
LIN {X 0,Y 473.847,Z 674.331,A -85,B 0,C 180,E1 -7187.145,E2 -7187.145} C_VEL
LIN {X 0,Y 473.994,Z 669.26,A -85,B 0,C 180,E1 -7188.886,E2 -7188.886} C_VEL
LIN {X 0,Y 474.258,Z 662.738,A -85,B 0,C 180,E1 -7190.618,E2 -7190.618} C_VEL
LIN {X 0,Y 474.631,Z 655.701,A -85,B 0,C 180,E1 -7192.127,E2 -7192.127} C_VEL
LIN {X 0,Y 475.087,Z 647.254,A -85,B 0,C 180,E1 -7193.63,E2 -7193.63} C_VEL
LIN {X 0,Y 475.652,Z 637.127,A -85,B 0,C 180,E1 -7195.126,E2 -7195.126} C_VEL
LIN {X 0,Y 476.251,Z 626.809,A -85,B 0,C 180,E1 -7196.404,E2 -7196.404} C_VEL
LIN {X 0,Y 476.977,Z 614.469,A -85,B 0,C 180,E1 -7197.678,E2 -7197.678} C_VEL
LIN {X 0,Y 477.748,Z 601.588,A -85,B 0,C 180,E1 -7198.778,E2 -7198.778} C_VEL
LIN {X 0,Y 478.433,Z 588.991,A -85,B 0,C 180,E1 -7199.668,E2 -7199.668} C_VEL
LIN {X 0,Y 479.127,Z 574.88,A -85,B 0,C 180,E1 -7200.473,E2 -7200.473} C_VEL
LIN {X 0,Y 479.686,Z 560.767,A -85,B 0,C 180,E1 -7201.102,E2 -7201.102} C_VEL
LIN {X 0,Y 480.167,Z 545.652,A -85,B 0,C 180,E1 -7201.599,E2 -7201.599} C_VEL
LIN {X 0,Y 480.45,Z 530.006,A -85,B 0,C 180,E1 -7201.938,E2 -7201.938} C_VEL
LIN {X 0,Y 482.22,Z 413.113,A -85,B 0,C 180,E1 -7203.883,E2 -7203.883} C_VEL
LIN {X 0,Y 482.487,Z 390.756,A -85,B 0,C 180,E1 -7204.277,E2 -7204.277} C_VEL
LIN {X 0,Y 478.355,Z 373.136,A -85,B 0,C 180,E1 -7204.848,E2 -7204.848} C_VEL
LIN {X 0,Y 477.198,Z 366.337,A -85,B 0,C 180,E1 -7206.129,E2 -7206.129} C_VEL
LIN {X 0,Y 474.705,Z 355.982,A -85,B 0,C 180,E1 -7208.219,E2 -7208.219} C_VEL
LIN {X 0,Y 474.679,Z 355.982,A -85,B 0,C 180,E1 -7211.097,E2 -7211.097} C_VEL
LIN {X 0,Y 474.642,Z 355.987,A -85,B 0,C 180,E1 -7213.704,E2 -7213.704} C_VEL
LIN {X 0,Y 474.642,Z 355.991,A -85,B 0,C 180,E1 -7216.34,E2 -7216.34} C_VEL
LIN {X 0,Y 474.666,Z 355.984,A -85,B 0,C 180,E1 -7219.01,E2 -7219.01} C_VEL
LIN {X 0,Y 474.593,Z 355.991,A -85,B 0,C 180,E1 -7221.729,E2 -7221.729} C_VEL
LIN {X 0,Y 474.629,Z 355.991,A -85,B 0,C 180,E1 -7224.494,E2 -7224.494} C_VEL
LIN {X 0,Y 474.601,Z 355.99,A -85,B 0,C 180,E1 -7227.326,E2 -7227.326} C_VEL
LIN {X 0,Y 474.598,Z 355.995,A -85,B 0,C 180,E1 -7230.23,E2 -7230.23} C_VEL
LIN {X 0,Y 474.618,Z 355.987,A -85,B 0,C 180,E1 -7233.222,E2 -7233.222} C_VEL
LIN {X 0,Y 474.572,Z 355.998,A -85,B 0,C 180,E1 -7236.325,E2 -7236.325} C_VEL
LIN {X 0,Y 474.604,Z 355.99,A -85,B 0,C 180,E1 -7239.55,E2 -7239.55} C_VEL
LIN {X 0,Y 474.567,Z 355.993,A -85,B 0,C 180,E1 -7242.939,E2 -7242.939} C_VEL
LIN {X 0,Y 474.6,Z 355.993,A -85,B 0,C 180,E1 -7245.893,E2 -7245.893} C_VEL
LIN {X 0,Y 474.582,Z 355.991,A -85,B 0,C 180,E1 -7249.047,E2 -7249.047} C_VEL
LIN {X 0,Y 474.588,Z 355.995,A -85,B 0,C 180,E1 -7251.707,E2 -7251.707} C_VEL
LIN {X 0,Y 474.604,Z 355.993,A -85,B 0,C 180,E1 -7254.723,E2 -7254.723} C_VEL
LIN {X 0,Y 474.616,Z 355.997,A -85,B 0,C 180,E1 -7257.785,E2 -7257.785} C_VEL
LIN {X 0,Y 474.65,Z 356.173,A -85,B 0,C 180,E1 -7259.772,E2 -7259.772} C_VEL
LIN {X 0,Y 477.98,Z 369.765,A -85,B 0,C 180,E1 -7262.171,E2 -7262.171} C_VEL
LIN {X 0,Y 479.109,Z 375.636,A -85,B 0,C 180,E1 -7263.148,E2 -7263.148} C_VEL
LIN {X 0,Y 477.979,Z 396.063,A -85,B 0,C 180,E1 -7266.161,E2 -7266.161} C_VEL
LIN {X 0,Y 482.381,Z 420.157,A -85,B 0,C 180,E1 -7266.851,E2 -7266.851} C_VEL
LIN {X 0,Y 480.45,Z 547.435,A -85,B 0,C 180,E1 -7268.97,E2 -7268.97} C_VEL
LIN {X 0,Y 480.095,Z 567.459,A -85,B 0,C 180,E1 -7269.346,E2 -7269.346} C_VEL
LIN {X 0,Y 479.577,Z 582.602,A -85,B 0,C 180,E1 -7269.799,E2 -7269.799} C_VEL
LIN {X 0,Y 478.991,Z 596.882,A -85,B 0,C 180,E1 -7270.388,E2 -7270.388} C_VEL
LIN {X 0,Y 478.314,Z 610.998,A -85,B 0,C 180,E1 -7271.139,E2 -7271.139} C_VEL
LIN {X 0,Y 477.529,Z 625.467,A -85,B 0,C 180,E1 -7272.107,E2 -7272.107} C_VEL
LIN {X 0,Y 476.822,Z 638.391,A -85,B 0,C 180,E1 -7273.167,E2 -7273.167} C_VEL
LIN {X 0,Y 476.065,Z 650.596,A -85,B 0,C 180,E1 -7274.369,E2 -7274.369} C_VEL
LIN {X 0,Y 475.487,Z 661.59,A -85,B 0,C 180,E1 -7275.665,E2 -7275.665} C_VEL
LIN {X 0,Y 474.897,Z 672.286,A -85,B 0,C 180,E1 -7277.173,E2 -7277.173} C_VEL
LIN {X 0,Y 474.492,Z 681.169,A -85,B 0,C 180,E1 -7278.681,E2 -7278.681} C_VEL
LIN {X 0,Y 474.134,Z 688.549,A -85,B 0,C 180,E1 -7280.184,E2 -7280.184} C_VEL
LIN {X 0,Y 473.948,Z 695.377,A -85,B 0,C 180,E1 -7281.901,E2 -7281.901} C_VEL
LIN {X 0,Y 473.815,Z 700.72,A -85,B 0,C 180,E1 -7283.614,E2 -7283.614} C_VEL
LIN {X 0,Y 473.78,Z 703.792,A -85,B 0,C 180,E1 -7284.893,E2 -7284.893} C_VEL
LIN {X 0,Y 473.744,Z 706.805,A -85,B 0,C 180,E1 -7286.597,E2 -7286.597} C_VEL
LIN {X 0,Y 473.721,Z 708.606,A -85,B 0,C 180,E1 -7288.298,E2 -7288.298} C_VEL
LIN {X 0,Y 473.666,Z 709.233,A -85,B 0,C 180,E1 -7289.999,E2 -7289.999} C_VEL
LIN {X 0,Y 473.721,Z 708.639,A -85,B 0,C 180,E1 -7291.699,E2 -7291.699} C_VEL
LIN {X 0,Y 473.777,Z 706.871,A -85,B 0,C 180,E1 -7293.4,E2 -7293.4} C_VEL
LIN {X 0,Y 473.782,Z 703.901,A -85,B 0,C 180,E1 -7295.105,E2 -7295.105} C_VEL
LIN {X 0,Y 473.892,Z 699.662,A -85,B 0,C 180,E1 -7296.812,E2 -7296.812} C_VEL
LIN {X 0,Y 474.008,Z 694.036,A -85,B 0,C 180,E1 -7298.525,E2 -7298.525} C_VEL
LIN {X 0,Y 474.242,Z 686.872,A -85,B 0,C 180,E1 -7300.242,E2 -7300.242} C_VEL
LIN {X 0,Y 474.627,Z 679.205,A -85,B 0,C 180,E1 -7301.746,E2 -7301.746} C_VEL
LIN {X 0,Y 475.064,Z 669.961,A -85,B 0,C 180,E1 -7303.255,E2 -7303.255} C_VEL
LIN {X 0,Y 475.611,Z 660.511,A -85,B 0,C 180,E1 -7304.547,E2 -7304.547} C_VEL
LIN {X 0,Y 476.348,Z 648.33,A -85,B 0,C 180,E1 -7305.948,E2 -7305.948} C_VEL
LIN {X 0,Y 477.048,Z 635.88,A -85,B 0,C 180,E1 -7307.135,E2 -7307.135} C_VEL
LIN {X 0,Y 477.844,Z 622.144,A -85,B 0,C 180,E1 -7308.211,E2 -7308.211} C_VEL
LIN {X 0,Y 478.592,Z 608.673,A -85,B 0,C 180,E1 -7309.069,E2 -7309.069} C_VEL
LIN {X 0,Y 479.277,Z 594.706,A -85,B 0,C 180,E1 -7309.779,E2 -7309.779} C_VEL
LIN {X 0,Y 479.84,Z 579.917,A -85,B 0,C 180,E1 -7310.355,E2 -7310.355} C_VEL
LIN {X 0,Y 480.301,Z 564.316,A -85,B 0,C 180,E1 -7310.782,E2 -7310.782} C_VEL
LIN {X 0,Y 482.259,Z 418.99,A -85,B 0,C 180,E1 -7313.152,E2 -7313.152} C_VEL
LIN {X 0,Y 478.002,Z 397.184,A -85,B 0,C 180,E1 -7313.744,E2 -7313.744} C_VEL
LIN {X 0,Y 479.127,Z 376.783,A -85,B 0,C 180,E1 -7316.702,E2 -7316.702} C_VEL
LIN {X 0,Y 478.672,Z 372.955,A -85,B 0,C 180,E1 -7317.302,E2 -7317.302} C_VEL
LIN {X 0,Y 475.255,Z 358.585,A -85,B 0,C 180,E1 -7319.698,E2 -7319.698} C_VEL
LIN {X 0,Y 474.66,Z 355.987,A -85,B 0,C 180,E1 -7320.164,E2 -7320.164} C_VEL
LIN {X 0,Y 474.616,Z 355.988,A -85,B 0,C 180,E1 -7323.22,E2 -7323.22} C_VEL
LIN {X 0,Y 474.571,Z 355.997,A -85,B 0,C 180,E1 -7326.323,E2 -7326.323} C_VEL
LIN {X 0,Y 474.59,Z 355.992,A -85,B 0,C 180,E1 -7329.642,E2 -7329.642} C_VEL
LIN {X 0,Y 474.577,Z 355.998,A -85,B 0,C 180,E1 -7332.231,E2 -7332.231} C_VEL
LIN {X 0,Y 474.604,Z 355.986,A -85,B 0,C 180,E1 -7335.297,E2 -7335.297} C_VEL
LIN {X 0,Y 474.582,Z 355.997,A -85,B 0,C 180,E1 -7338.211,E2 -7338.211} C_VEL
LIN {X 0,Y 474.605,Z 355.991,A -85,B 0,C 180,E1 -7340.45,E2 -7340.45} C_VEL
LIN {X 0,Y 474.56,Z 355.994,A -85,B 0,C 180,E1 -7343.674,E2 -7343.674} C_VEL
LIN {X 0,Y 474.621,Z 355.985,A -85,B 0,C 180,E1 -7346.778,E2 -7346.778} C_VEL
LIN {X 0,Y 474.582,Z 355.993,A -85,B 0,C 180,E1 -7349.768,E2 -7349.768} C_VEL
LIN {X 0,Y 474.587,Z 355.99,A -85,B 0,C 180,E1 -7352.684,E2 -7352.684} C_VEL
LIN {X 0,Y 474.611,Z 355.987,A -85,B 0,C 180,E1 -7355.505,E2 -7355.505} C_VEL
LIN {X 0,Y 474.619,Z 355.985,A -85,B 0,C 180,E1 -7358.884,E2 -7358.884} C_VEL
LIN {X 0,Y 474.617,Z 355.99,A -85,B 0,C 180,E1 -7361.883,E2 -7361.883} C_VEL
LIN {X 0,Y 474.672,Z 355.98,A -85,B 0,C 180,E1 -7364.544,E2 -7364.544} C_VEL
LIN {X 0,Y 474.689,Z 355.984,A -85,B 0,C 180,E1 -7368.037,E2 -7368.037} C_VEL
LIN {X 0,Y 474.68,Z 355.979,A -85,B 0,C 180,E1 -7371.486,E2 -7371.486} C_VEL
LIN {X 0,Y 474.726,Z 355.98,A -85,B 0,C 180,E1 -7374.052,E2 -7374.052} C_VEL
LIN {X 0,Y 474.856,Z 355.957,A -85,B 0,C 180,E1 -7377.455,E2 -7377.455} C_VEL
LIN {X 0,Y 474.864,Z 355.963,A -85,B 0,C 180,E1 -7380,E2 -7380} C_VEL
LIN {X 0,Y 474.855,Z 355.957,A -85,B 0,C 180,E1 -7382.545,E2 -7382.545} C_VEL
LIN {X 0,Y 474.721,Z 355.98,A -85,B 0,C 180,E1 -7385.949,E2 -7385.949} C_VEL
LIN {X 0,Y 474.679,Z 355.979,A -85,B 0,C 180,E1 -7388.515,E2 -7388.515} C_VEL
LIN {X 0,Y 474.678,Z 355.986,A -85,B 0,C 180,E1 -7391.963,E2 -7391.963} C_VEL
LIN {X 0,Y 474.673,Z 355.98,A -85,B 0,C 180,E1 -7395.457,E2 -7395.457} C_VEL
LIN {X 0,Y 474.644,Z 355.981,A -85,B 0,C 180,E1 -7399.011,E2 -7399.011} C_VEL
LIN {X 0,Y 474.573,Z 355.996,A -85,B 0,C 180,E1 -7401.73,E2 -7401.73} C_VEL
LIN {X 0,Y 474.612,Z 355.987,A -85,B 0,C 180,E1 -7404.496,E2 -7404.496} C_VEL
LIN {X 0,Y 474.584,Z 355.99,A -85,B 0,C 180,E1 -7407.328,E2 -7407.328} C_VEL
LIN {X 0,Y 474.584,Z 355.993,A -85,B 0,C 180,E1 -7410.232,E2 -7410.232} C_VEL
LIN {X 0,Y 474.614,Z 355.986,A -85,B 0,C 180,E1 -7413.223,E2 -7413.223} C_VEL
LIN {X 0,Y 474.562,Z 355.994,A -85,B 0,C 180,E1 -7416.326,E2 -7416.326} C_VEL
LIN {X 0,Y 474.59,Z 355.994,A -85,B 0,C 180,E1 -7419.645,E2 -7419.645} C_VEL
